Yaskawa INFORM job: DEMO_ROOF_SIDE_0625_3PAINT_25.JBI

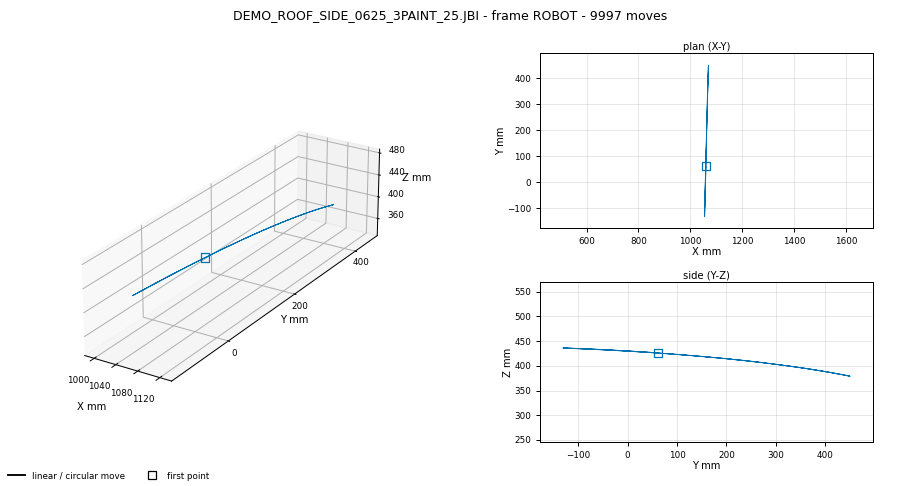
[picture p0: tool path of DEMO_ROOF_SIDE_0625_3PAINT_25.JBI in frame ROBOT, 9997 of 9997 moves have a stored position in this frame; points joined in program order, loops and branches not executed]
/JOB
//NAME DEMO_ROOF_SIDE_0625_3PAINT25
//POS
///NPOS 9997,0,0,0,0,0
///TOOL 0
///USER 0
///POSTYPE ROBOT
///RECTAN
///RCONF 1,0,0,0,0,0,0,0,0,0,0,0,0,0,0,0,0,0,0,0,0,0,0,0
C00000=1059.838,61.557,426.310,171.754,29.522,155.486
C00001=1059.832,61.309,426.327,171.753,29.519,155.486
C00002=1059.826,61.059,426.345,171.752,29.517,155.485
C00003=1059.820,60.810,426.362,171.750,29.515,155.485
C00004=1059.814,60.561,426.379,171.748,29.512,155.485
C00005=1059.807,60.311,426.396,171.747,29.509,155.484
C00006=1059.801,60.062,426.413,171.746,29.507,155.484
C00007=1059.795,59.813,426.431,171.744,29.505,155.484
C00008=1059.789,59.563,426.447,171.743,29.502,155.483
C00009=1059.783,59.314,426.465,171.741,29.500,155.483
C00010=1059.777,59.065,426.482,171.739,29.497,155.482
C00011=1059.771,58.816,426.499,171.739,29.494,155.482
C00012=1059.765,58.566,426.517,171.737,29.492,155.482
C00013=1059.758,58.317,426.534,171.735,29.489,155.481
C00014=1059.752,58.067,426.550,171.733,29.487,155.481
C00015=1059.746,57.818,426.568,171.733,29.485,155.481
C00016=1059.740,57.569,426.585,171.731,29.482,155.480
C00017=1059.734,57.319,426.602,171.729,29.479,155.480
C00018=1059.728,57.070,426.619,171.728,29.477,155.480
C00019=1059.722,56.821,426.635,171.726,29.474,155.479
C00020=1059.716,56.571,426.653,171.725,29.472,155.479
C00021=1059.710,56.322,426.670,171.723,29.470,155.478
C00022=1059.703,56.072,426.687,171.722,29.467,155.478
C00023=1059.698,55.823,426.704,171.720,29.464,155.478
C00024=1059.692,55.574,426.721,171.719,29.462,155.477
C00025=1059.685,55.324,426.738,171.718,29.459,155.477
C00026=1059.680,55.075,426.755,171.716,29.457,155.477
C00027=1059.673,54.826,426.772,171.714,29.454,155.476
C00028=1059.666,54.577,426.789,171.712,29.452,155.476
C00029=1059.661,54.327,426.806,171.712,29.449,155.475
C00030=1059.655,54.078,426.823,171.710,29.446,155.475
C00031=1059.648,53.828,426.839,171.708,29.444,155.475
C00032=1059.643,53.579,426.857,171.707,29.441,155.474
C00033=1059.637,53.330,426.873,171.706,29.439,155.474
C00034=1059.631,53.081,426.890,171.704,29.437,155.474
C00035=1059.625,52.831,426.907,171.703,29.434,155.473
C00036=1059.619,52.582,426.924,171.701,29.431,155.473
C00037=1059.613,52.333,426.941,171.700,29.429,155.473
C00038=1059.607,52.083,426.959,171.698,29.426,155.472
C00039=1059.601,51.834,426.975,171.697,29.424,155.472
C00040=1059.595,51.584,426.991,171.695,29.422,155.472
C00041=1059.589,51.335,427.009,171.693,29.419,155.471
C00042=1059.583,51.085,427.025,171.693,29.416,155.471
C00043=1059.576,50.836,427.042,171.691,29.413,155.470
C00044=1059.571,50.587,427.059,171.689,29.411,155.470
C00045=1059.565,50.338,427.076,171.688,29.409,155.470
C00046=1059.558,50.088,427.093,171.687,29.406,155.469
C00047=1059.553,49.838,427.110,171.685,29.404,155.469
C00048=1059.547,49.590,427.127,171.683,29.401,155.469
C00049=1059.541,49.340,427.143,171.682,29.398,155.468
C00050=1059.534,49.091,427.160,171.680,29.396,155.468
C00051=1059.529,48.841,427.177,171.679,29.394,155.467
C00052=1059.523,48.592,427.193,171.678,29.391,155.467
C00053=1059.517,48.343,427.210,171.676,29.388,155.467
C00054=1059.511,48.093,427.227,171.674,29.386,155.466
C00055=1059.505,47.843,427.244,171.674,29.383,155.466
C00056=1059.499,47.595,427.261,171.672,29.381,155.466
C00057=1059.493,47.345,427.277,171.670,29.378,155.465
C00058=1059.487,47.096,427.294,171.668,29.376,155.465
C00059=1059.481,46.847,427.311,171.668,29.373,155.464
C00060=1059.475,46.597,427.327,171.666,29.370,155.464
C00061=1059.468,46.313,427.346,171.664,29.368,155.464
C00062=1059.462,46.027,427.366,171.663,29.365,155.463
C00063=1059.455,45.742,427.385,171.661,29.361,155.463
C00064=1059.448,45.458,427.404,171.659,29.359,155.462
C00065=1059.442,45.208,427.420,171.658,29.356,155.462
C00066=1059.436,44.959,427.437,171.656,29.354,155.462
C00067=1059.430,44.709,427.453,171.654,29.351,155.461
C00068=1059.424,44.461,427.470,171.654,29.348,155.461
C00069=1059.419,44.211,427.487,171.652,29.346,155.461
C00070=1059.412,43.961,427.503,171.650,29.343,155.460
C00071=1059.406,43.711,427.520,171.649,29.341,155.460
C00072=1059.401,43.462,427.536,171.648,29.338,155.459
C00073=1059.394,43.213,427.553,171.646,29.336,155.459
C00074=1059.388,42.964,427.569,171.645,29.333,155.459
C00075=1059.382,42.715,427.585,171.643,29.331,155.458
C00076=1059.376,42.465,427.602,171.641,29.328,155.458
C00077=1059.370,42.215,427.618,171.640,29.326,155.458
C00078=1059.364,41.966,427.635,171.639,29.324,155.457
C00079=1059.358,41.717,427.651,171.637,29.321,155.457
C00080=1059.352,41.468,427.668,171.635,29.319,155.457
C00081=1059.346,41.218,427.684,171.635,29.316,155.456
C00082=1059.340,40.969,427.700,171.633,29.313,155.456
C00083=1059.333,40.719,427.717,171.631,29.311,155.455
C00084=1059.327,40.470,427.733,171.630,29.308,155.455
C00085=1059.322,40.220,427.750,171.628,29.306,155.455
C00086=1059.316,39.971,427.766,171.627,29.304,155.454
C00087=1059.310,39.721,427.783,171.625,29.301,155.454
C00088=1059.304,39.472,427.799,171.624,29.299,155.454
C00089=1059.298,39.223,427.815,171.622,29.296,155.453
C00090=1059.292,38.973,427.831,171.620,29.293,155.453
C00091=1059.286,38.724,427.848,171.620,29.291,155.453
C00092=1059.280,38.474,427.864,171.618,29.288,155.452
C00093=1059.274,38.225,427.880,171.616,29.286,155.452
C00094=1059.268,37.975,427.897,171.615,29.283,155.452
C00095=1059.262,37.726,427.913,171.614,29.281,155.451
C00096=1059.255,37.477,427.929,171.612,29.279,155.451
C00097=1059.249,37.228,427.945,171.610,29.276,155.450
C00098=1059.243,36.978,427.961,171.609,29.274,155.450
C00099=1059.237,36.729,427.977,171.607,29.271,155.450
C00100=1059.231,36.479,427.994,171.606,29.269,155.449
C00101=1059.224,36.230,428.010,171.605,29.266,155.449
C00102=1059.218,35.980,428.026,171.603,29.264,155.449
C00103=1059.212,35.731,428.042,171.601,29.261,155.448
C00104=1059.206,35.482,428.058,171.600,29.259,155.448
C00105=1059.200,35.232,428.075,171.599,29.256,155.448
C00106=1059.194,34.983,428.090,171.597,29.254,155.447
C00107=1059.188,34.734,428.107,171.595,29.252,155.447
C00108=1059.182,34.484,428.122,171.594,29.249,155.447
C00109=1059.176,34.235,428.138,171.593,29.247,155.446
C00110=1059.170,33.985,428.155,171.591,29.244,155.446
C00111=1059.164,33.736,428.170,171.590,29.242,155.446
C00112=1059.158,33.487,428.187,171.588,29.239,155.445
C00113=1059.152,33.238,428.203,171.586,29.237,155.445
C00114=1059.146,32.988,428.219,171.586,29.234,155.445
C00115=1059.139,32.738,428.235,171.584,29.232,155.444
C00116=1059.133,32.488,428.251,171.582,29.229,155.444
C00117=1059.127,32.239,428.267,171.580,29.227,155.444
C00118=1059.121,31.990,428.283,171.579,29.224,155.443
C00119=1059.115,31.740,428.299,171.578,29.222,155.443
C00120=1059.108,31.491,428.314,171.576,29.220,155.443
C00121=1059.103,31.241,428.331,171.575,29.217,155.442
C00122=1059.097,30.992,428.347,171.573,29.215,155.442
C00123=1059.091,30.743,428.363,171.571,29.212,155.442
C00124=1059.085,30.493,428.379,171.571,29.210,155.441
C00125=1059.078,30.209,428.397,171.569,29.207,155.441
C00126=1059.071,29.923,428.415,171.567,29.204,155.440
C00127=1059.064,29.639,428.434,171.565,29.201,155.440
C00128=1059.057,29.354,428.451,171.563,29.199,155.440
C00129=1059.051,29.105,428.468,171.562,29.196,155.439
C00130=1059.045,28.855,428.483,171.561,29.194,155.439
C00131=1059.039,28.606,428.499,171.559,29.191,155.439
C00132=1059.033,28.356,428.515,171.557,29.189,155.438
C00133=1059.027,28.106,428.531,171.556,29.186,155.438
C00134=1059.020,27.857,428.546,171.555,29.184,155.438
C00135=1059.014,27.608,428.562,171.553,29.181,155.437
C00136=1059.009,27.358,428.578,171.551,29.179,155.437
C00137=1059.002,27.109,428.594,171.550,29.177,155.437
C00138=1058.996,26.860,428.610,171.548,29.174,155.436
C00139=1058.990,26.610,428.625,171.547,29.172,155.436
C00140=1058.984,26.361,428.641,171.546,29.169,155.436
C00141=1058.977,26.111,428.657,171.544,29.167,155.435
C00142=1058.971,25.862,428.672,171.542,29.164,155.435
C00143=1058.965,25.612,428.689,171.541,29.162,155.435
C00144=1058.959,25.363,428.704,171.540,29.160,155.434
C00145=1058.953,25.113,428.720,171.538,29.158,155.434
C00146=1058.946,24.864,428.735,171.536,29.155,155.434
C00147=1058.941,24.614,428.751,171.535,29.153,155.433
C00148=1058.935,24.366,428.766,171.533,29.150,155.433
C00149=1058.929,24.116,428.782,171.532,29.148,155.432
C00150=1058.922,23.867,428.797,171.531,29.146,155.432
C00151=1058.917,23.617,428.813,171.529,29.143,155.432
C00152=1058.910,23.368,428.829,171.527,29.141,155.432
C00153=1058.904,23.118,428.844,171.526,29.138,155.431
C00154=1058.898,22.869,428.860,171.525,29.136,155.431
C00155=1058.892,22.619,428.875,171.523,29.134,155.431
C00156=1058.886,22.369,428.892,171.522,29.131,155.430
C00157=1058.880,22.120,428.907,171.520,29.129,155.430
C00158=1058.874,21.870,428.923,171.518,29.126,155.430
C00159=1058.868,21.622,428.937,171.517,29.124,155.429
C00160=1058.862,21.372,428.954,171.516,29.122,155.429
C00161=1058.856,21.123,428.969,171.514,29.119,155.429
C00162=1058.850,20.873,428.985,171.512,29.117,155.428
C00163=1058.843,20.624,429.000,171.511,29.114,155.428
C00164=1058.837,20.374,429.016,171.509,29.112,155.428
C00165=1058.831,20.125,429.031,171.508,29.109,155.427
C00166=1058.825,19.875,429.046,171.507,29.107,155.427
C00167=1058.819,19.626,429.062,171.505,29.105,155.427
C00168=1058.813,19.377,429.077,171.503,29.102,155.426
C00169=1058.807,19.127,429.093,171.502,29.100,155.426
C00170=1058.801,18.878,429.108,171.501,29.098,155.426
C00171=1058.794,18.628,429.123,171.499,29.095,155.425
C00172=1058.788,18.379,429.139,171.497,29.093,155.425
C00173=1058.782,18.129,429.154,171.496,29.090,155.425
C00174=1058.776,17.879,429.170,171.494,29.088,155.424
C00175=1058.770,17.631,429.185,171.493,29.086,155.424
C00176=1058.764,17.381,429.200,171.492,29.083,155.424
C00177=1058.758,17.131,429.216,171.490,29.081,155.423
C00178=1058.751,16.882,429.231,171.488,29.079,155.423
C00179=1058.745,16.632,429.246,171.487,29.076,155.423
C00180=1058.739,16.382,429.262,171.485,29.074,155.422
C00181=1058.733,16.134,429.277,171.484,29.071,155.422
C00182=1058.728,15.884,429.293,171.482,29.069,155.422
C00183=1058.721,15.634,429.307,171.481,29.067,155.421
C00184=1058.715,15.385,429.322,171.479,29.064,155.421
C00185=1058.709,15.135,429.339,171.477,29.062,155.421
C00186=1058.703,14.886,429.353,171.477,29.060,155.420
C00187=1058.697,14.637,429.368,171.475,29.057,155.420
C00188=1058.691,14.387,429.384,171.473,29.055,155.420
C00189=1058.684,14.104,429.401,171.472,29.052,155.419
C00190=1058.676,13.820,429.419,171.470,29.050,155.419
C00191=1058.669,13.537,429.435,171.468,29.047,155.419
C00192=1058.662,13.253,429.453,171.467,29.044,155.418
C00193=1058.656,13.004,429.468,171.465,29.042,155.418
C00194=1058.650,12.754,429.483,171.463,29.040,155.418
C00195=1058.644,12.504,429.498,171.462,29.037,155.417
C00196=1058.637,12.255,429.513,171.460,29.035,155.417
C00197=1058.631,12.005,429.528,171.458,29.033,155.417
C00198=1058.625,11.756,429.543,171.457,29.031,155.417
C00199=1058.619,11.507,429.558,171.456,29.028,155.416
C00200=1058.613,11.257,429.573,171.454,29.026,155.416
C00201=1058.606,11.007,429.588,171.452,29.023,155.416
C00202=1058.600,10.758,429.603,171.451,29.021,155.415
C00203=1058.594,10.509,429.618,171.449,29.019,155.415
C00204=1058.588,10.259,429.633,171.447,29.016,155.415
C00205=1058.581,10.010,429.648,171.447,29.014,155.414
C00206=1058.576,9.760,429.663,171.445,29.012,155.414
C00207=1058.570,9.511,429.678,171.443,29.010,155.414
C00208=1058.563,9.262,429.693,171.442,29.007,155.413
C00209=1058.557,9.012,429.708,171.440,29.005,155.413
C00210=1058.551,8.762,429.723,171.438,29.003,155.413
C00211=1058.545,8.513,429.738,171.437,29.001,155.413
C00212=1058.538,8.264,429.753,171.436,28.999,155.412
C00213=1058.532,8.014,429.768,171.434,28.996,155.412
C00214=1058.526,7.764,429.783,171.432,28.994,155.412
C00215=1058.520,7.515,429.797,171.431,28.991,155.411
C00216=1058.514,7.265,429.813,171.429,28.989,155.411
C00217=1058.508,7.016,429.828,171.428,28.987,155.411
C00218=1058.502,6.767,429.842,171.427,28.984,155.410
C00219=1058.496,6.517,429.857,171.425,28.982,155.410
C00220=1058.489,6.267,429.872,171.423,28.980,155.410
C00221=1058.483,6.018,429.887,171.421,28.978,155.410
C00222=1058.477,5.769,429.902,171.420,28.975,155.409
C00223=1058.471,5.519,429.917,171.418,28.973,155.409
C00224=1058.464,5.270,429.932,171.417,28.971,155.409
C00225=1058.459,5.020,429.946,171.416,28.969,155.408
C00226=1058.452,4.770,429.961,171.414,28.966,155.408
C00227=1058.446,4.521,429.976,171.412,28.964,155.408
C00228=1058.440,4.272,429.990,171.411,28.961,155.407
C00229=1058.434,4.022,430.005,171.409,28.959,155.407
C00230=1058.428,3.772,430.021,171.408,28.957,155.407
C00231=1058.422,3.523,430.035,171.407,28.954,155.406
C00232=1058.416,3.273,430.050,171.405,28.952,155.406
C00233=1058.410,3.025,430.065,171.403,28.950,155.406
C00234=1058.404,2.775,430.080,171.401,28.948,155.406
C00235=1058.398,2.525,430.094,171.400,28.945,155.405
C00236=1058.392,2.276,430.108,171.398,28.943,155.405
C00237=1058.386,2.026,430.123,171.397,28.941,155.405
C00238=1058.379,1.776,430.138,171.396,28.939,155.404
C00239=1058.374,1.527,430.153,171.394,28.936,155.404
C00240=1058.367,1.278,430.168,171.392,28.934,155.404
C00241=1058.362,1.028,430.182,171.391,28.931,155.403
C00242=1058.355,0.778,430.197,171.389,28.929,155.403
C00243=1058.349,0.529,430.212,171.387,28.927,155.403
C00244=1058.343,0.280,430.226,171.386,28.925,155.403
C00245=1058.337,0.030,430.241,171.385,28.922,155.402
C00246=1058.331,-0.219,430.255,171.383,28.920,155.402
C00247=1058.325,-0.469,430.270,171.381,28.918,155.402
C00248=1058.319,-0.718,430.285,171.380,28.915,155.401
C00249=1058.313,-0.968,430.299,171.378,28.913,155.401
C00250=1058.307,-1.217,430.313,171.376,28.910,155.401
C00251=1058.301,-1.467,430.328,171.376,28.908,155.400
C00252=1058.294,-1.717,430.343,171.374,28.906,155.400
C00253=1058.288,-1.998,430.360,171.372,28.903,155.400
C00254=1058.281,-2.280,430.376,171.371,28.901,155.400
C00255=1058.275,-2.561,430.392,171.368,28.898,155.399
C00256=1058.268,-2.843,430.409,171.366,28.896,155.399
C00257=1058.262,-3.092,430.423,171.365,28.893,155.398
C00258=1058.256,-3.342,430.438,171.364,28.891,155.398
C00259=1058.250,-3.592,430.452,171.362,28.889,155.398
C00260=1058.243,-3.841,430.466,171.361,28.887,155.398
C00261=1058.237,-4.091,430.481,171.359,28.885,155.397
C00262=1058.231,-4.340,430.495,171.357,28.882,155.397
C00263=1058.225,-4.590,430.510,171.356,28.880,155.397
C00264=1058.219,-4.839,430.523,171.354,28.878,155.397
C00265=1058.212,-5.089,430.538,171.352,28.876,155.396
C00266=1058.206,-5.339,430.553,171.351,28.874,155.396
C00267=1058.200,-5.588,430.567,171.350,28.872,155.396
C00268=1058.193,-5.837,430.582,171.348,28.869,155.395
C00269=1058.188,-6.087,430.595,171.346,28.867,155.395
C00270=1058.181,-6.336,430.610,171.345,28.865,155.395
C00271=1058.175,-6.586,430.624,171.343,28.863,155.395
C00272=1058.169,-6.835,430.639,171.341,28.860,155.394
C00273=1058.163,-7.085,430.652,171.339,28.858,155.394
C00274=1058.156,-7.334,430.667,171.338,28.856,155.394
C00275=1058.151,-7.584,430.681,171.337,28.854,155.394
C00276=1058.144,-7.834,430.696,171.335,28.852,155.393
C00277=1058.138,-8.083,430.709,171.334,28.850,155.393
C00278=1058.132,-8.332,430.724,171.332,28.847,155.393
C00279=1058.126,-8.582,430.738,171.330,28.845,155.392
C00280=1058.119,-8.831,430.752,171.329,28.843,155.392
C00281=1058.114,-9.081,430.766,171.327,28.841,155.392
C00282=1058.107,-9.331,430.781,171.325,28.839,155.392
C00283=1058.102,-9.580,430.795,171.323,28.836,155.391
C00284=1058.095,-9.830,430.809,171.323,28.834,155.391
C00285=1058.089,-10.079,430.823,171.321,28.832,155.391
C00286=1058.083,-10.329,430.838,171.319,28.830,155.390
C00287=1058.077,-10.578,430.851,171.318,28.828,155.390
C00288=1058.070,-10.828,430.866,171.316,28.825,155.390
C00289=1058.065,-11.077,430.880,171.314,28.823,155.390
C00290=1058.058,-11.327,430.894,171.313,28.821,155.389
C00291=1058.052,-11.576,430.908,171.311,28.819,155.389
C00292=1058.047,-11.826,430.922,171.309,28.817,155.389
C00293=1058.040,-12.075,430.936,171.308,28.815,155.389
C00294=1058.034,-12.325,430.950,171.307,28.812,155.388
C00295=1058.027,-12.575,430.964,171.305,28.810,155.388
C00296=1058.021,-12.824,430.978,171.303,28.808,155.388
C00297=1058.016,-13.073,430.992,171.302,28.806,155.387
C00298=1058.009,-13.323,431.006,171.300,28.804,155.387
C00299=1058.003,-13.572,431.021,171.298,28.801,155.387
C00300=1057.997,-13.822,431.035,171.297,28.799,155.387
C00301=1057.991,-14.072,431.048,171.295,28.797,155.387
C00302=1057.985,-14.321,431.063,171.293,28.795,155.386
C00303=1057.979,-14.571,431.077,171.292,28.793,155.386
C00304=1057.973,-14.820,431.090,171.291,28.791,155.386
C00305=1057.967,-15.070,431.105,171.289,28.789,155.385
C00306=1057.960,-15.319,431.118,171.287,28.787,155.385
C00307=1057.955,-15.569,431.132,171.286,28.784,155.385
C00308=1057.948,-15.819,431.146,171.284,28.782,155.385
C00309=1057.942,-16.068,431.160,171.282,28.780,155.384
C00310=1057.936,-16.318,431.174,171.281,28.778,155.384
C00311=1057.929,-16.567,431.187,171.279,28.776,155.384
C00312=1057.923,-16.817,431.202,171.277,28.774,155.384
C00313=1057.917,-17.066,431.215,171.275,28.772,155.383
C00314=1057.911,-17.315,431.229,171.275,28.770,155.383
C00315=1057.904,-17.565,431.243,171.273,28.767,155.383
C00316=1057.899,-17.815,431.257,171.271,28.766,155.383
C00317=1057.893,-18.069,431.271,171.270,28.764,155.382
C00318=1057.886,-18.325,431.285,171.268,28.761,155.382
C00319=1057.879,-18.579,431.299,171.266,28.759,155.382
C00320=1057.873,-18.833,431.313,171.265,28.757,155.382
C00321=1057.867,-19.083,431.326,171.263,28.755,155.381
C00322=1057.861,-19.333,431.341,171.261,28.753,155.381
C00323=1057.855,-19.582,431.354,171.259,28.751,155.381
C00324=1057.849,-19.832,431.368,171.258,28.749,155.381
C00325=1057.842,-20.082,431.381,171.256,28.746,155.380
C00326=1057.836,-20.331,431.395,171.254,28.744,155.380
C00327=1057.830,-20.580,431.409,171.253,28.743,155.380
C00328=1057.824,-20.830,431.423,171.251,28.740,155.380
C00329=1057.818,-21.079,431.437,171.250,28.738,155.379
C00330=1057.812,-21.329,431.450,171.248,28.736,155.379
C00331=1057.805,-21.579,431.464,171.247,28.734,155.379
C00332=1057.800,-21.828,431.478,171.245,28.732,155.379
C00333=1057.793,-22.078,431.491,171.243,28.730,155.378
C00334=1057.787,-22.328,431.504,171.242,28.728,155.378
C00335=1057.781,-22.577,431.518,171.240,28.726,155.378
C00336=1057.775,-22.826,431.532,171.238,28.724,155.378
C00337=1057.769,-23.076,431.545,171.236,28.722,155.377
C00338=1057.763,-23.326,431.559,171.235,28.719,155.377
C00339=1057.756,-23.575,431.572,171.233,28.717,155.377
C00340=1057.751,-23.825,431.586,171.231,28.715,155.377
C00341=1057.745,-24.074,431.599,171.230,28.713,155.376
C00342=1057.738,-24.324,431.613,171.228,28.711,155.376
C00343=1057.732,-24.574,431.627,171.226,28.709,155.376
C00344=1057.726,-24.823,431.640,171.226,28.707,155.376
C00345=1057.720,-25.072,431.654,171.224,28.705,155.375
C00346=1057.714,-25.322,431.668,171.222,28.703,155.375
C00347=1057.708,-25.572,431.681,171.220,28.701,155.375
C00348=1057.701,-25.821,431.694,171.219,28.699,155.375
C00349=1057.696,-26.070,431.708,171.217,28.697,155.375
C00350=1057.689,-26.320,431.722,171.215,28.695,155.374
C00351=1057.683,-26.570,431.735,171.214,28.693,155.374
C00352=1057.677,-26.819,431.749,171.212,28.690,155.374
C00353=1057.671,-27.069,431.762,171.210,28.689,155.374
C00354=1057.665,-27.318,431.775,171.208,28.686,155.373
C00355=1057.659,-27.568,431.788,171.207,28.685,155.373
C00356=1057.652,-27.818,431.802,171.205,28.683,155.373
C00357=1057.646,-28.067,431.815,171.203,28.680,155.373
C00358=1057.640,-28.316,431.828,171.202,28.679,155.372
C00359=1057.634,-28.566,431.842,171.200,28.677,155.372
C00360=1057.628,-28.816,431.855,171.198,28.675,155.372
C00361=1057.621,-29.090,431.870,171.196,28.673,155.372
C00362=1057.614,-29.365,431.885,171.195,28.670,155.372
C00363=1057.607,-29.640,431.899,171.193,28.668,155.371
C00364=1057.599,-29.916,431.914,171.191,28.666,155.371
C00365=1057.594,-30.166,431.927,171.190,28.664,155.371
C00366=1057.588,-30.415,431.940,171.188,28.662,155.371
C00367=1057.582,-30.664,431.953,171.186,28.660,155.370
C00368=1057.576,-30.914,431.967,171.185,28.658,155.370
C00369=1057.569,-31.164,431.980,171.183,28.656,155.370
C00370=1057.563,-31.413,431.993,171.181,28.654,155.370
C00371=1057.557,-31.663,432.006,171.179,28.652,155.369
C00372=1057.550,-31.912,432.019,171.178,28.651,155.369
C00373=1057.545,-32.162,432.032,171.176,28.648,155.369
C00374=1057.538,-32.411,432.045,171.174,28.647,155.369
C00375=1057.532,-32.661,432.059,171.173,28.644,155.369
C00376=1057.526,-32.911,432.073,171.171,28.642,155.368
C00377=1057.520,-33.161,432.085,171.169,28.641,155.368
C00378=1057.514,-33.410,432.099,171.167,28.638,155.368
C00379=1057.508,-33.659,432.112,171.166,28.637,155.368
C00380=1057.502,-33.909,432.124,171.164,28.634,155.368
C00381=1057.494,-34.188,432.140,171.162,28.632,155.367
C00382=1057.487,-34.467,432.154,171.161,28.631,155.367
C00383=1057.481,-34.747,432.168,171.159,28.628,155.367
C00384=1057.474,-35.026,432.183,171.157,28.626,155.367
C00385=1057.468,-35.275,432.196,171.156,28.624,155.366
C00386=1057.461,-35.525,432.209,171.154,28.622,155.366
C00387=1057.455,-35.775,432.223,171.152,28.620,155.366
C00388=1057.449,-36.025,432.235,171.150,28.618,155.366
C00389=1057.443,-36.274,432.248,171.149,28.616,155.365
C00390=1057.437,-36.524,432.261,171.147,28.615,155.365
C00391=1057.431,-36.773,432.274,171.145,28.612,155.365
C00392=1057.425,-37.022,432.288,171.143,28.611,155.365
C00393=1057.419,-37.272,432.300,171.142,28.608,155.365
C00394=1057.413,-37.522,432.314,171.140,28.607,155.364
C00395=1057.407,-37.772,432.327,171.138,28.605,155.364
C00396=1057.401,-38.021,432.340,171.137,28.603,155.364
C00397=1057.395,-38.271,432.352,171.135,28.601,155.364
C00398=1057.389,-38.520,432.366,171.133,28.599,155.364
C00399=1057.383,-38.770,432.378,171.131,28.597,155.363
C00400=1057.376,-39.020,432.391,171.130,28.595,155.363
C00401=1057.370,-39.269,432.404,171.128,28.594,155.363
C00402=1057.363,-39.519,432.417,171.126,28.591,155.363
C00403=1057.357,-39.769,432.430,171.125,28.590,155.363
C00404=1057.351,-40.018,432.443,171.123,28.588,155.362
C00405=1057.345,-40.267,432.455,171.121,28.586,155.362
C00406=1057.338,-40.517,432.468,171.119,28.584,155.362
C00407=1057.333,-40.767,432.481,171.118,28.583,155.362
C00408=1057.327,-41.016,432.493,171.116,28.580,155.362
C00409=1057.320,-41.266,432.506,171.114,28.579,155.362
C00410=1057.314,-41.516,432.519,171.112,28.577,155.361
C00411=1057.308,-41.765,432.532,171.111,28.575,155.361
C00412=1057.302,-42.014,432.544,171.109,28.573,155.361
C00413=1057.296,-42.264,432.557,171.107,28.571,155.361
C00414=1057.289,-42.514,432.570,171.106,28.569,155.361
C00415=1057.284,-42.763,432.583,171.104,28.568,155.360
C00416=1057.277,-43.012,432.595,171.102,28.566,155.360
C00417=1057.271,-43.262,432.608,171.100,28.564,155.360
C00418=1057.265,-43.512,432.620,171.099,28.562,155.360
C00419=1057.259,-43.761,432.634,171.097,28.560,155.360
C00420=1057.252,-44.011,432.646,171.095,28.558,155.359
C00421=1057.246,-44.261,432.658,171.093,28.557,155.359
C00422=1057.240,-44.510,432.671,171.092,28.555,155.359
C00423=1057.234,-44.760,432.684,171.090,28.553,155.359
C00424=1057.228,-45.010,432.697,171.088,28.551,155.359
C00425=1057.221,-45.259,432.709,171.087,28.549,155.359
C00426=1057.215,-45.509,432.722,171.085,28.548,155.358
C00427=1057.209,-45.759,432.734,171.083,28.546,155.358
C00428=1057.203,-46.009,432.747,171.081,28.544,155.358
C00429=1057.196,-46.257,432.760,171.080,28.542,155.358
C00430=1057.190,-46.507,432.772,171.078,28.541,155.358
C00431=1057.185,-46.757,432.785,171.076,28.538,155.357
C00432=1057.179,-47.007,432.797,171.074,28.537,155.357
C00433=1057.172,-47.256,432.810,171.073,28.535,155.357
C00434=1057.166,-47.506,432.823,171.071,28.533,155.357
C00435=1057.160,-47.756,432.835,171.069,28.531,155.357
C00436=1057.154,-48.006,432.848,171.067,28.530,155.357
C00437=1057.147,-48.255,432.860,171.066,28.528,155.356
C00438=1057.142,-48.504,432.872,171.064,28.526,155.356
C00439=1057.136,-48.754,432.885,171.062,28.524,155.356
C00440=1057.130,-49.004,432.898,171.061,28.522,155.356
C00441=1057.123,-49.253,432.910,171.059,28.521,155.356
C00442=1057.117,-49.503,432.922,171.057,28.519,155.356
C00443=1057.111,-49.752,432.935,171.055,28.517,155.355
C00444=1057.104,-50.002,432.947,171.054,28.515,155.355
C00445=1057.098,-50.282,432.961,171.052,28.514,155.355
C00446=1057.091,-50.561,432.975,171.050,28.511,155.355
C00447=1057.084,-50.842,432.989,171.047,28.509,155.355
C00448=1057.077,-51.121,433.003,171.046,28.508,155.354
C00449=1057.071,-51.370,433.015,171.044,28.506,155.354
C00450=1057.065,-51.620,433.027,171.042,28.505,155.354
C00451=1057.058,-51.870,433.039,171.040,28.503,155.354
C00452=1057.052,-52.120,433.052,171.039,28.501,155.354
C00453=1057.045,-52.369,433.064,171.037,28.500,155.354
C00454=1057.039,-52.619,433.076,171.035,28.498,155.354
C00455=1057.033,-52.869,433.088,171.033,28.496,155.353
C00456=1057.026,-53.118,433.100,171.032,28.495,155.353
C00457=1057.021,-53.367,433.112,171.030,28.493,155.353
C00458=1057.014,-53.617,433.124,171.028,28.491,155.353
C00459=1057.008,-53.867,433.137,171.027,28.490,155.353
C00460=1057.002,-54.116,433.149,171.025,28.488,155.353
C00461=1056.995,-54.366,433.161,171.023,28.486,155.353
C00462=1056.989,-54.616,433.173,171.021,28.485,155.352
C00463=1056.982,-54.865,433.185,171.020,28.483,155.352
C00464=1056.977,-55.115,433.198,171.018,28.481,155.352
C00465=1056.971,-55.364,433.209,171.015,28.480,155.352
C00466=1056.964,-55.614,433.221,171.013,28.478,155.352
C00467=1056.958,-55.864,433.234,171.012,28.476,155.352
C00468=1056.951,-56.113,433.246,171.010,28.475,155.352
C00469=1056.945,-56.363,433.258,171.008,28.473,155.351
C00470=1056.939,-56.613,433.270,171.006,28.471,155.351
C00471=1056.932,-56.862,433.282,171.005,28.470,155.351
C00472=1056.927,-57.111,433.295,171.003,28.468,155.351
C00473=1056.920,-57.361,433.307,171.001,28.466,155.351
C00474=1056.914,-57.611,433.318,170.999,28.465,155.351
C00475=1056.908,-57.861,433.330,170.997,28.464,155.351
C00476=1056.901,-58.111,433.342,170.996,28.462,155.350
C00477=1056.895,-58.360,433.354,170.994,28.460,155.350
C00478=1056.889,-58.609,433.366,170.992,28.459,155.350
C00479=1056.883,-58.859,433.378,170.990,28.457,155.350
C00480=1056.877,-59.109,433.391,170.989,28.455,155.350
C00481=1056.870,-59.358,433.403,170.987,28.454,155.350
C00482=1056.864,-59.608,433.414,170.985,28.452,155.350
C00483=1056.858,-59.858,433.426,170.984,28.451,155.349
C00484=1056.852,-60.107,433.438,170.982,28.449,155.349
C00485=1056.845,-60.357,433.450,170.980,28.448,155.349
C00486=1056.840,-60.606,433.462,170.978,28.446,155.349
C00487=1056.834,-60.856,433.474,170.976,28.445,155.349
C00488=1056.827,-61.106,433.486,170.975,28.443,155.349
C00489=1056.821,-61.356,433.498,170.972,28.441,155.349
C00490=1056.815,-61.605,433.510,170.970,28.439,155.349
C00491=1056.809,-61.855,433.521,170.969,28.438,155.348
C00492=1056.803,-62.105,433.534,170.967,28.436,155.348
C00493=1056.796,-62.354,433.546,170.965,28.435,155.348
C00494=1056.790,-62.603,433.557,170.963,28.433,155.348
C00495=1056.784,-62.854,433.569,170.961,28.432,155.348
C00496=1056.778,-63.103,433.581,170.960,28.430,155.348
C00497=1056.771,-63.353,433.593,170.958,28.428,155.348
C00498=1056.765,-63.602,433.604,170.956,28.427,155.347
C00499=1056.759,-63.852,433.616,170.954,28.426,155.347
C00500=1056.753,-64.102,433.628,170.953,28.424,155.347
C00501=1056.747,-64.351,433.640,170.951,28.422,155.347
C00502=1056.741,-64.601,433.652,170.949,28.421,155.347
C00503=1056.735,-64.851,433.664,170.947,28.419,155.347
C00504=1056.728,-65.100,433.675,170.946,28.418,155.347
C00505=1056.723,-65.350,433.687,170.944,28.416,155.347
C00506=1056.716,-65.600,433.699,170.942,28.415,155.347
C00507=1056.710,-65.849,433.710,170.940,28.413,155.346
C00508=1056.704,-66.099,433.722,170.938,28.411,155.346
C00509=1056.697,-66.380,433.735,170.936,28.410,155.346
C00510=1056.690,-66.660,433.749,170.934,28.408,155.346
C00511=1056.683,-66.942,433.762,170.932,28.406,155.346
C00512=1056.676,-67.223,433.775,170.930,28.404,155.346
C00513=1056.671,-67.472,433.787,170.928,28.403,155.346
C00514=1056.665,-67.722,433.798,170.926,28.402,155.346
C00515=1056.658,-67.972,433.810,170.924,28.400,155.345
C00516=1056.652,-68.221,433.821,170.923,28.398,155.345
C00517=1056.646,-68.471,433.834,170.921,28.397,155.345
C00518=1056.641,-68.721,433.845,170.919,28.396,155.345
C00519=1056.634,-68.970,433.856,170.917,28.394,155.345
C00520=1056.628,-69.220,433.868,170.916,28.392,155.345
C00521=1056.622,-69.470,433.880,170.914,28.391,155.345
C00522=1056.616,-69.720,433.891,170.912,28.390,155.345
C00523=1056.610,-69.969,433.903,170.910,28.388,155.344
C00524=1056.604,-70.219,433.914,170.909,28.386,155.344
C00525=1056.598,-70.468,433.926,170.906,28.385,155.344
C00526=1056.592,-70.718,433.937,170.904,28.383,155.344
C00527=1056.586,-70.967,433.949,170.902,28.382,155.344
C00528=1056.580,-71.217,433.960,170.900,28.381,155.344
C00529=1056.574,-71.467,433.973,170.899,28.379,155.344
C00530=1056.568,-71.717,433.984,170.897,28.377,155.344
C00531=1056.561,-71.966,433.996,170.895,28.376,155.344
C00532=1056.555,-72.216,434.007,170.893,28.375,155.344
C00533=1056.549,-72.465,434.018,170.892,28.373,155.343
C00534=1056.544,-72.715,434.030,170.890,28.371,155.343
C00535=1056.537,-72.965,434.041,170.888,28.370,155.343
C00536=1056.531,-73.214,434.053,170.886,28.369,155.343
C00537=1056.525,-73.464,434.064,170.885,28.367,155.343
C00538=1056.519,-73.714,434.075,170.883,28.366,155.343
C00539=1056.513,-73.964,434.087,170.881,28.364,155.343
C00540=1056.508,-74.213,434.098,170.878,28.363,155.343
C00541=1056.501,-74.463,434.110,170.876,28.361,155.343
C00542=1056.495,-74.712,434.121,170.875,28.360,155.343
C00543=1056.489,-74.962,434.132,170.873,28.359,155.342
C00544=1056.482,-75.212,434.144,170.871,28.358,155.342
C00545=1056.477,-75.462,434.155,170.869,28.356,155.342
C00546=1056.470,-75.712,434.167,170.868,28.355,155.342
C00547=1056.465,-75.961,434.177,170.866,28.353,155.342
C00548=1056.458,-76.211,434.189,170.864,28.352,155.342
C00549=1056.451,-76.460,434.200,170.862,28.350,155.342
C00550=1056.445,-76.710,434.211,170.860,28.349,155.342
C00551=1056.439,-76.959,434.222,170.859,28.348,155.342
C00552=1056.433,-77.209,434.234,170.857,28.347,155.342
C00553=1056.427,-77.459,434.245,170.854,28.345,155.342
C00554=1056.421,-77.709,434.256,170.852,28.344,155.342
C00555=1056.415,-77.958,434.267,170.851,28.342,155.341
C00556=1056.408,-78.208,434.279,170.849,28.341,155.341
C00557=1056.402,-78.457,434.290,170.847,28.340,155.341
C00558=1056.396,-78.708,434.301,170.845,28.338,155.341
C00559=1056.390,-78.957,434.312,170.843,28.337,155.341
C00560=1056.384,-79.206,434.323,170.842,28.336,155.341
C00561=1056.378,-79.456,434.335,170.840,28.335,155.341
C00562=1056.372,-79.706,434.345,170.838,28.334,155.341
C00563=1056.366,-79.956,434.357,170.836,28.332,155.341
C00564=1056.359,-80.205,434.367,170.833,28.331,155.341
C00565=1056.353,-80.455,434.378,170.832,28.330,155.341
C00566=1056.347,-80.704,434.390,170.830,28.328,155.341
C00567=1056.341,-80.954,434.401,170.828,28.327,155.341
C00568=1056.334,-81.203,434.411,170.826,28.326,155.341
C00569=1056.328,-81.454,434.423,170.824,28.325,155.341
C00570=1056.322,-81.703,434.433,170.823,28.323,155.340
C00571=1056.316,-81.953,434.445,170.821,28.322,155.340
C00572=1056.309,-82.203,434.455,170.819,28.321,155.340
C00573=1056.302,-82.487,434.468,170.816,28.320,155.340
C00574=1056.295,-82.769,434.480,170.815,28.318,155.340
C00575=1056.288,-83.052,434.492,170.813,28.317,155.340
C00576=1056.281,-83.336,434.505,170.810,28.315,155.340
C00577=1056.275,-83.585,434.516,170.808,28.314,155.340
C00578=1056.268,-83.835,434.527,170.806,28.313,155.340
C00579=1056.263,-84.084,434.538,170.805,28.312,155.340
C00580=1056.256,-84.334,434.548,170.803,28.311,155.340
C00581=1056.250,-84.584,434.560,170.801,28.309,155.340
C00582=1056.244,-84.833,434.570,170.799,28.308,155.340
C00583=1056.237,-85.083,434.581,170.796,28.307,155.340
C00584=1056.231,-85.333,434.592,170.795,28.306,155.340
C00585=1056.225,-85.582,434.603,170.793,28.305,155.340
C00586=1056.219,-85.832,434.614,170.791,28.304,155.340
C00587=1056.213,-86.082,434.624,170.789,28.302,155.340
C00588=1056.207,-86.332,434.635,170.787,28.301,155.340
C00589=1056.201,-86.582,434.646,170.786,28.300,155.339
C00590=1056.194,-86.831,434.656,170.784,28.299,155.339
C00591=1056.188,-87.081,434.667,170.782,28.298,155.339
C00592=1056.182,-87.331,434.678,170.780,28.297,155.339
C00593=1056.176,-87.580,434.688,170.777,28.295,155.339
C00594=1056.169,-87.830,434.700,170.776,28.294,155.339
C00595=1056.164,-88.080,434.711,170.774,28.293,155.339
C00596=1056.157,-88.329,434.721,170.772,28.292,155.339
C00597=1056.151,-88.579,434.732,170.770,28.291,155.339
C00598=1056.145,-88.828,434.743,170.768,28.289,155.339
C00599=1056.139,-89.078,434.753,170.766,28.288,155.339
C00600=1056.133,-89.328,434.764,170.765,28.287,155.339
C00601=1056.127,-89.578,434.775,170.763,28.286,155.339
C00602=1056.120,-89.827,434.785,170.760,28.285,155.339
C00603=1056.114,-90.077,434.796,170.758,28.284,155.339
C00604=1056.108,-90.326,434.806,170.756,28.283,155.339
C00605=1056.102,-90.576,434.817,170.755,28.281,155.339
C00606=1056.096,-90.827,434.828,170.753,28.280,155.339
C00607=1056.089,-91.076,434.838,170.751,28.279,155.339
C00608=1056.084,-91.325,434.849,170.749,28.278,155.339
C00609=1056.078,-91.575,434.860,170.747,28.277,155.339
C00610=1056.071,-91.825,434.871,170.746,28.276,155.339
C00611=1056.065,-92.075,434.881,170.744,28.275,155.339
C00612=1056.060,-92.324,434.892,170.741,28.274,155.339
C00613=1056.053,-92.574,434.902,170.739,28.273,155.339
C00614=1056.047,-92.824,434.913,170.737,28.271,155.339
C00615=1056.041,-93.074,434.923,170.735,28.270,155.339
C00616=1056.035,-93.323,434.934,170.734,28.269,155.339
C00617=1056.029,-93.573,434.944,170.732,28.268,155.339
C00618=1056.022,-93.822,434.955,170.730,28.267,155.339
C00619=1056.017,-94.073,434.965,170.728,28.266,155.338
C00620=1056.010,-94.322,434.976,170.726,28.265,155.338
C00621=1056.004,-94.571,434.986,170.724,28.264,155.338
C00622=1055.999,-94.821,434.997,170.722,28.263,155.338
C00623=1055.992,-95.071,435.007,170.720,28.262,155.338
C00624=1055.986,-95.321,435.018,170.718,28.261,155.338
C00625=1055.980,-95.570,435.028,170.716,28.260,155.338
C00626=1055.974,-95.820,435.039,170.714,28.258,155.338
C00627=1055.968,-96.069,435.049,170.713,28.257,155.338
C00628=1055.962,-96.320,435.059,170.711,28.256,155.338
C00629=1055.956,-96.569,435.070,170.709,28.255,155.338
C00630=1055.949,-96.819,435.081,170.706,28.254,155.338
C00631=1055.944,-97.069,435.091,170.704,28.253,155.338
C00632=1055.938,-97.318,435.101,170.703,28.252,155.338
C00633=1055.931,-97.568,435.112,170.701,28.251,155.338
C00634=1055.925,-97.818,435.122,170.699,28.250,155.338
C00635=1055.919,-98.067,435.133,170.697,28.249,155.338
C00636=1055.913,-98.317,435.142,170.695,28.248,155.338
C00637=1055.906,-98.603,435.155,170.692,28.247,155.338
C00638=1055.899,-98.888,435.166,170.691,28.246,155.338
C00639=1055.892,-99.173,435.178,170.688,28.245,155.338
C00640=1055.885,-99.459,435.190,170.686,28.244,155.338
C00641=1055.879,-99.709,435.199,170.684,28.243,155.338
C00642=1055.872,-99.958,435.209,170.682,28.242,155.338
C00643=1055.866,-100.208,435.221,170.680,28.242,155.338
C00644=1055.860,-100.458,435.230,170.679,28.240,155.338
C00645=1055.854,-100.708,435.240,170.676,28.239,155.338
C00646=1055.848,-100.957,435.251,170.674,28.238,155.338
C00647=1055.842,-101.207,435.260,170.672,28.238,155.338
C00648=1055.835,-101.456,435.271,170.670,28.237,155.338
C00649=1055.830,-101.706,435.281,170.668,28.236,155.338
C00650=1055.823,-101.956,435.291,170.667,28.235,155.338
C00651=1055.817,-102.206,435.301,170.665,28.234,155.338
C00652=1055.811,-102.456,435.312,170.663,28.233,155.338
C00653=1055.805,-102.705,435.321,170.660,28.232,155.338
C00654=1055.798,-102.955,435.332,170.658,28.231,155.338
C00655=1055.793,-103.205,435.342,170.656,28.230,155.338
C00656=1055.787,-103.455,435.351,170.655,28.230,155.338
C00657=1055.780,-103.704,435.362,170.653,28.229,155.338
C00658=1055.773,-103.954,435.372,170.651,28.228,155.338
C00659=1055.768,-104.204,435.383,170.649,28.227,155.339
C00660=1055.762,-104.453,435.392,170.647,28.226,155.338
C00661=1055.755,-104.703,435.402,170.644,28.225,155.338
C00662=1055.750,-104.953,435.413,170.642,28.224,155.339
C00663=1055.743,-105.203,435.422,170.641,28.223,155.339
C00664=1055.737,-105.452,435.432,170.639,28.223,155.339
C00665=1055.731,-105.702,435.442,170.637,28.222,155.339
C00666=1055.725,-105.952,435.452,170.635,28.221,155.339
C00667=1055.719,-106.201,435.462,170.633,28.220,155.339
C00668=1055.713,-106.451,435.472,170.631,28.219,155.339
C00669=1055.707,-106.700,435.482,170.629,28.218,155.339
C00670=1055.701,-106.951,435.492,170.627,28.217,155.339
C00671=1055.695,-107.200,435.502,170.625,28.217,155.339
C00672=1055.688,-107.450,435.512,170.623,28.216,155.339
C00673=1055.682,-107.700,435.521,170.621,28.215,155.339
C00674=1055.676,-107.950,435.531,170.619,28.214,155.339
C00675=1055.670,-108.199,435.542,170.617,28.214,155.339
C00676=1055.664,-108.449,435.551,170.615,28.213,155.339
C00677=1055.657,-108.699,435.561,170.613,28.212,155.339
C00678=1055.651,-108.949,435.571,170.611,28.211,155.339
C00679=1055.645,-109.198,435.581,170.609,28.211,155.339
C00680=1055.639,-109.448,435.590,170.607,28.210,155.339
C00681=1055.632,-109.697,435.600,170.605,28.209,155.339
C00682=1055.626,-109.947,435.610,170.603,28.209,155.339
C00683=1055.621,-110.197,435.620,170.602,28.208,155.339
C00684=1055.614,-110.447,435.630,170.599,28.207,155.339
C00685=1055.608,-110.696,435.640,170.597,28.206,155.339
C00686=1055.602,-110.946,435.649,170.595,28.205,155.339
C00687=1055.596,-111.196,435.659,170.593,28.205,155.339
C00688=1055.590,-111.446,435.668,170.591,28.204,155.339
C00689=1055.583,-111.696,435.678,170.589,28.203,155.340
C00690=1055.577,-111.945,435.688,170.587,28.202,155.340
C00691=1055.571,-112.195,435.698,170.585,28.202,155.340
C00692=1055.565,-112.444,435.707,170.583,28.201,155.340
C00693=1055.558,-112.694,435.717,170.581,28.200,155.340
C00694=1055.553,-112.944,435.727,170.579,28.200,155.340
C00695=1055.547,-113.194,435.737,170.577,28.199,155.340
C00696=1055.541,-113.444,435.746,170.575,28.198,155.340
C00697=1055.535,-113.694,435.756,170.573,28.198,155.340
C00698=1055.528,-113.943,435.765,170.571,28.197,155.340
C00699=1055.522,-114.193,435.775,170.569,28.196,155.340
C00700=1055.516,-114.442,435.785,170.567,28.195,155.340
C00701=1055.509,-114.727,435.795,170.565,28.195,155.340
C00702=1055.502,-115.010,435.806,170.562,28.194,155.340
C00703=1055.495,-115.295,435.818,170.560,28.193,155.340
C00704=1055.488,-115.579,435.828,170.558,28.193,155.340
C00705=1055.482,-115.829,435.838,170.555,28.192,155.341
C00706=1055.476,-116.078,435.847,170.554,28.191,155.341
C00707=1055.470,-116.328,435.857,170.552,28.191,155.341
C00708=1055.464,-116.578,435.866,170.550,28.190,155.341
C00709=1055.457,-116.828,435.876,170.548,28.190,155.341
C00710=1055.452,-117.077,435.885,170.546,28.189,155.341
C00711=1055.446,-117.327,435.895,170.544,28.188,155.341
C00712=1055.440,-117.576,435.904,170.541,28.187,155.341
C00713=1055.433,-117.826,435.913,170.539,28.187,155.341
C00714=1055.426,-118.076,435.923,170.538,28.186,155.341
C00715=1055.420,-118.326,435.932,170.536,28.186,155.341
C00716=1055.414,-118.575,435.942,170.534,28.185,155.341
C00717=1055.408,-118.825,435.951,170.532,28.184,155.341
C00718=1055.402,-119.075,435.961,170.530,28.184,155.341
C00719=1055.396,-119.325,435.970,170.527,28.183,155.342
C00720=1055.390,-119.574,435.980,170.525,28.183,155.342
C00721=1055.384,-119.824,435.989,170.523,28.182,155.342
C00722=1055.378,-120.074,435.998,170.521,28.182,155.342
C00723=1055.371,-120.324,436.007,170.520,28.181,155.342
C00724=1055.365,-120.573,436.017,170.518,28.180,155.342
C00725=1055.359,-120.823,436.026,170.516,28.180,155.342
C00726=1055.353,-121.073,436.036,170.513,28.179,155.342
C00727=1055.347,-121.322,436.045,170.511,28.179,155.342
C00728=1055.341,-121.572,436.055,170.509,28.178,155.342
C00729=1055.335,-121.822,436.063,170.507,28.178,155.342
C00730=1055.329,-122.072,436.073,170.505,28.177,155.342
C00731=1055.322,-122.322,436.082,170.503,28.177,155.342
C00732=1055.316,-122.571,436.092,170.502,28.177,155.343
C00733=1055.310,-122.820,436.101,170.499,28.176,155.343
C00734=1055.304,-123.071,436.110,170.497,28.175,155.343
C00735=1055.298,-123.321,436.119,170.495,28.175,155.343
C00736=1055.292,-123.570,436.129,170.493,28.174,155.343
C00737=1055.285,-123.820,436.138,170.491,28.174,155.343
C00738=1055.279,-124.070,436.147,170.489,28.174,155.343
C00739=1055.274,-124.319,436.156,170.487,28.173,155.343
C00740=1055.267,-124.569,436.165,170.485,28.173,155.343
C00741=1055.261,-124.819,436.175,170.483,28.172,155.343
C00742=1055.255,-125.069,436.183,170.481,28.171,155.344
C00743=1055.248,-125.319,436.193,170.479,28.171,155.344
C00744=1055.243,-125.568,436.202,170.477,28.171,155.344
C00745=1055.236,-125.818,436.211,170.475,28.170,155.344
C00746=1055.230,-126.068,436.220,170.473,28.170,155.344
C00747=1055.224,-126.318,436.229,170.470,28.170,155.344
C00748=1055.218,-126.568,436.239,170.468,28.169,155.344
C00749=1055.212,-126.817,436.247,170.466,28.169,155.344
C00750=1055.206,-127.067,436.256,170.464,28.168,155.344
C00751=1055.199,-127.317,436.266,170.462,28.168,155.344
C00752=1055.193,-127.567,436.274,170.461,28.167,155.345
C00753=1055.187,-127.816,436.283,170.459,28.167,155.345
C00754=1055.182,-128.066,436.293,170.457,28.166,155.345
C00755=1055.178,-128.316,436.303,170.455,28.165,155.345
C00756=1055.175,-128.566,436.314,170.453,28.163,155.344
C00757=1055.174,-128.817,436.325,170.452,28.161,155.344
C00758=1055.174,-129.067,436.338,170.450,28.157,155.344
C00759=1055.174,-129.318,436.351,170.449,28.154,155.343
C00760=1055.176,-129.567,436.364,170.448,28.150,155.343
C00761=1055.179,-129.819,436.379,170.447,28.145,155.342
C00762=1055.184,-130.070,436.394,170.447,28.140,155.341
C00763=1055.190,-130.321,436.410,170.445,28.135,155.340
C00764=1055.196,-130.571,436.427,170.445,28.128,155.339
C00765=1054.825,-130.594,436.216,170.397,28.295,155.372
C00766=1054.818,-130.344,436.200,170.399,28.301,155.373
C00767=1054.813,-130.093,436.184,170.399,28.307,155.374
C00768=1054.808,-129.843,436.169,170.399,28.312,155.375
C00769=1054.804,-129.591,436.155,170.400,28.316,155.376
C00770=1054.802,-129.341,436.141,170.401,28.320,155.376
C00771=1054.801,-129.091,436.128,170.402,28.324,155.377
C00772=1054.802,-128.840,436.116,170.404,28.327,155.377
C00773=1054.804,-128.590,436.104,170.405,28.329,155.378
C00774=1054.806,-128.339,436.093,170.407,28.331,155.378
C00775=1054.810,-128.089,436.083,170.409,28.333,155.378
C00776=1054.815,-127.840,436.073,170.411,28.333,155.378
C00777=1054.821,-127.589,436.064,170.413,28.334,155.378
C00778=1054.828,-127.340,436.055,170.415,28.334,155.378
C00779=1054.833,-127.091,436.046,170.417,28.335,155.378
C00780=1054.839,-126.840,436.037,170.419,28.335,155.377
C00781=1054.846,-126.591,436.028,170.421,28.336,155.377
C00782=1054.852,-126.341,436.018,170.423,28.336,155.377
C00783=1054.858,-126.091,436.010,170.425,28.336,155.377
C00784=1054.863,-125.841,436.000,170.427,28.336,155.377
C00785=1054.870,-125.592,435.991,170.429,28.337,155.377
C00786=1054.876,-125.342,435.983,170.431,28.337,155.377
C00787=1054.882,-125.092,435.973,170.433,28.338,155.377
C00788=1054.889,-124.842,435.964,170.436,28.338,155.377
C00789=1054.895,-124.593,435.955,170.438,28.339,155.376
C00790=1054.901,-124.343,435.946,170.440,28.339,155.376
C00791=1054.907,-124.093,435.936,170.441,28.340,155.376
C00792=1054.913,-123.843,435.927,170.443,28.340,155.376
C00793=1054.920,-123.593,435.919,170.445,28.341,155.376
C00794=1054.925,-123.344,435.909,170.447,28.341,155.376
C00795=1054.931,-123.094,435.900,170.450,28.342,155.376
C00796=1054.938,-122.844,435.890,170.452,28.342,155.376
C00797=1054.944,-122.595,435.881,170.454,28.343,155.376
C00798=1054.950,-122.344,435.872,170.456,28.343,155.376
C00799=1054.957,-122.095,435.863,170.458,28.344,155.376
C00800=1054.962,-121.846,435.854,170.460,28.344,155.376
C00801=1054.968,-121.596,435.844,170.462,28.345,155.375
C00802=1054.974,-121.346,435.834,170.464,28.345,155.375
C00803=1054.981,-121.096,435.825,170.466,28.346,155.375
C00804=1054.987,-120.846,435.816,170.468,28.346,155.375
C00805=1054.993,-120.596,435.806,170.470,28.347,155.375
C00806=1054.998,-120.347,435.797,170.472,28.347,155.375
C00807=1055.005,-120.097,435.788,170.474,28.347,155.375
C00808=1055.011,-119.848,435.779,170.477,28.348,155.375
C00809=1055.018,-119.598,435.769,170.479,28.349,155.375
C00810=1055.024,-119.348,435.760,170.480,28.350,155.375
C00811=1055.030,-119.098,435.751,170.482,28.350,155.375
C00812=1055.036,-118.848,435.741,170.484,28.351,155.374
C00813=1055.042,-118.598,435.732,170.486,28.351,155.374
C00814=1055.047,-118.349,435.722,170.488,28.351,155.374
C00815=1055.054,-118.099,435.713,170.491,28.352,155.374
C00816=1055.060,-117.849,435.703,170.493,28.353,155.374
C00817=1055.067,-117.600,435.694,170.495,28.354,155.374
C00818=1055.073,-117.350,435.685,170.497,28.354,155.374
C00819=1055.079,-117.100,435.675,170.498,28.355,155.374
C00820=1055.085,-116.850,435.666,170.500,28.355,155.374
C00821=1055.091,-116.601,435.656,170.502,28.355,155.374
C00822=1055.098,-116.351,435.646,170.505,28.357,155.374
C00823=1055.104,-116.101,435.637,170.507,28.357,155.374
C00824=1055.110,-115.851,435.627,170.509,28.358,155.374
C00825=1055.116,-115.601,435.618,170.511,28.358,155.374
C00826=1055.123,-115.318,435.607,170.513,28.359,155.373
C00827=1055.130,-115.034,435.597,170.515,28.360,155.373
C00828=1055.137,-114.749,435.585,170.517,28.360,155.373
C00829=1055.144,-114.466,435.574,170.520,28.361,155.373
C00830=1055.150,-114.216,435.565,170.522,28.362,155.373
C00831=1055.156,-113.966,435.555,170.524,28.362,155.373
C00832=1055.162,-113.716,435.546,170.526,28.363,155.373
C00833=1055.169,-113.466,435.536,170.528,28.364,155.373
C00834=1055.175,-113.217,435.526,170.530,28.364,155.373
C00835=1055.180,-112.966,435.516,170.532,28.365,155.373
C00836=1055.186,-112.717,435.507,170.534,28.366,155.373
C00837=1055.192,-112.467,435.497,170.536,28.367,155.373
C00838=1055.199,-112.217,435.488,170.538,28.367,155.373
C00839=1055.205,-111.968,435.477,170.540,28.368,155.373
C00840=1055.211,-111.718,435.468,170.542,28.369,155.373
C00841=1055.217,-111.468,435.458,170.544,28.369,155.373
C00842=1055.224,-111.219,435.449,170.547,28.370,155.373
C00843=1055.230,-110.969,435.439,170.548,28.371,155.373
C00844=1055.236,-110.719,435.429,170.550,28.372,155.373
C00845=1055.242,-110.470,435.419,170.552,28.372,155.372
C00846=1055.248,-110.220,435.409,170.554,28.373,155.372
C00847=1055.254,-109.970,435.399,170.556,28.374,155.372
C00848=1055.260,-109.720,435.390,170.558,28.374,155.372
C00849=1055.266,-109.470,435.380,170.561,28.375,155.372
C00850=1055.273,-109.221,435.370,170.562,28.376,155.372
C00851=1055.279,-108.971,435.360,170.564,28.376,155.372
C00852=1055.285,-108.721,435.351,170.566,28.377,155.372
C00853=1055.291,-108.472,435.341,170.568,28.378,155.372
C00854=1055.297,-108.222,435.331,170.570,28.379,155.372
C00855=1055.303,-107.972,435.321,170.572,28.379,155.372
C00856=1055.309,-107.723,435.311,170.575,28.381,155.372
C00857=1055.316,-107.473,435.302,170.577,28.381,155.372
C00858=1055.322,-107.224,435.291,170.578,28.382,155.372
C00859=1055.328,-106.974,435.282,170.580,28.383,155.372
C00860=1055.334,-106.724,435.272,170.582,28.384,155.372
C00861=1055.340,-106.474,435.262,170.584,28.384,155.372
C00862=1055.346,-106.225,435.252,170.586,28.385,155.372
C00863=1055.353,-105.975,435.242,170.589,28.386,155.372
C00864=1055.359,-105.724,435.232,170.591,28.387,155.372
C00865=1055.365,-105.475,435.221,170.592,28.388,155.372
C00866=1055.371,-105.225,435.212,170.594,28.388,155.372
C00867=1055.377,-104.975,435.202,170.596,28.389,155.372
C00868=1055.383,-104.726,435.191,170.598,28.390,155.372
C00869=1055.389,-104.476,435.182,170.600,28.391,155.372
C00870=1055.396,-104.227,435.172,170.602,28.392,155.372
C00871=1055.401,-103.977,435.161,170.605,28.393,155.372
C00872=1055.407,-103.727,435.152,170.606,28.394,155.372
C00873=1055.414,-103.478,435.142,170.608,28.394,155.371
C00874=1055.419,-103.228,435.131,170.610,28.395,155.372
C00875=1055.426,-102.978,435.121,170.612,28.396,155.372
C00876=1055.433,-102.728,435.111,170.614,28.397,155.371
C00877=1055.439,-102.478,435.102,170.616,28.398,155.371
C00878=1055.444,-102.229,435.091,170.617,28.399,155.372
C00879=1055.451,-101.979,435.081,170.620,28.400,155.371
C00880=1055.457,-101.730,435.071,170.622,28.401,155.371
C00881=1055.463,-101.480,435.061,170.624,28.402,155.371
C00882=1055.469,-101.230,435.051,170.626,28.402,155.371
C00883=1055.476,-100.980,435.041,170.628,28.403,155.371
C00884=1055.482,-100.730,435.030,170.630,28.404,155.371
C00885=1055.488,-100.481,435.020,170.631,28.405,155.371
C00886=1055.494,-100.232,435.010,170.633,28.406,155.371
C00887=1055.500,-99.981,435.000,170.636,28.407,155.371
C00888=1055.506,-99.732,434.989,170.638,28.408,155.371
C00889=1055.512,-99.481,434.979,170.640,28.409,155.371
C00890=1055.520,-99.197,434.968,170.642,28.410,155.371
C00891=1055.527,-98.911,434.956,170.644,28.411,155.371
C00892=1055.534,-98.625,434.944,170.646,28.412,155.371
C00893=1055.541,-98.340,434.932,170.649,28.413,155.371
C00894=1055.547,-98.090,434.922,170.651,28.414,155.371
C00895=1055.553,-97.840,434.912,170.653,28.415,155.371
C00896=1055.559,-97.591,434.902,170.655,28.416,155.371
C00897=1055.565,-97.340,434.891,170.656,28.417,155.371
C00898=1055.572,-97.091,434.881,170.658,28.418,155.371
C00899=1055.577,-96.841,434.870,170.660,28.419,155.371
C00900=1055.584,-96.592,434.860,170.662,28.420,155.371
C00901=1055.590,-96.343,434.849,170.665,28.421,155.371
C00902=1055.595,-96.092,434.839,170.666,28.422,155.371
C00903=1055.602,-95.843,434.828,170.668,28.423,155.371
C00904=1055.608,-95.593,434.818,170.670,28.424,155.372
C00905=1055.614,-95.343,434.808,170.672,28.425,155.372
C00906=1055.620,-95.094,434.797,170.674,28.426,155.371
C00907=1055.625,-94.844,434.786,170.676,28.427,155.371
C00908=1055.632,-94.594,434.776,170.677,28.428,155.372
C00909=1055.638,-94.344,434.765,170.679,28.429,155.372
C00910=1055.644,-94.095,434.755,170.682,28.430,155.372
C00911=1055.650,-93.845,434.745,170.684,28.431,155.372
C00912=1055.656,-93.595,434.734,170.686,28.432,155.372
C00913=1055.663,-93.346,434.723,170.688,28.433,155.372
C00914=1055.668,-93.096,434.713,170.689,28.435,155.372
C00915=1055.675,-92.846,434.703,170.691,28.436,155.372
C00916=1055.680,-92.597,434.692,170.693,28.437,155.372
C00917=1055.687,-92.347,434.681,170.695,28.438,155.372
C00918=1055.693,-92.097,434.671,170.698,28.439,155.372
C00919=1055.699,-91.847,434.660,170.699,28.440,155.372
C00920=1055.706,-91.597,434.650,170.701,28.441,155.372
C00921=1055.711,-91.348,434.639,170.703,28.442,155.372
C00922=1055.717,-91.099,434.628,170.705,28.443,155.372
C00923=1055.724,-90.849,434.618,170.707,28.445,155.372
C00924=1055.730,-90.599,434.607,170.709,28.446,155.372
C00925=1055.735,-90.349,434.596,170.710,28.447,155.372
C00926=1055.742,-90.100,434.586,170.712,28.448,155.372
C00927=1055.748,-89.850,434.575,170.715,28.449,155.372
C00928=1055.754,-89.600,434.564,170.717,28.450,155.372
C00929=1055.760,-89.351,434.554,170.719,28.451,155.372
C00930=1055.767,-89.101,434.542,170.720,28.452,155.372
C00931=1055.772,-88.851,434.532,170.722,28.453,155.372
C00932=1055.779,-88.602,434.522,170.724,28.454,155.372
C00933=1055.785,-88.351,434.511,170.726,28.456,155.372
C00934=1055.791,-88.102,434.500,170.728,28.457,155.372
C00935=1055.797,-87.853,434.490,170.730,28.458,155.372
C00936=1055.804,-87.602,434.478,170.731,28.459,155.372
C00937=1055.809,-87.353,434.467,170.734,28.461,155.372
C00938=1055.816,-87.104,434.457,170.736,28.462,155.373
C00939=1055.822,-86.854,434.446,170.738,28.463,155.373
C00940=1055.828,-86.604,434.435,170.740,28.464,155.373
C00941=1055.834,-86.355,434.425,170.741,28.465,155.373
C00942=1055.841,-86.105,434.413,170.743,28.466,155.373
C00943=1055.846,-85.855,434.403,170.745,28.467,155.373
C00944=1055.853,-85.605,434.393,170.747,28.469,155.373
C00945=1055.859,-85.355,434.382,170.749,28.470,155.373
C00946=1055.865,-85.106,434.371,170.751,28.471,155.373
C00947=1055.872,-84.856,434.360,170.753,28.472,155.373
C00948=1055.878,-84.606,434.349,170.755,28.473,155.373
C00949=1055.884,-84.356,434.338,170.757,28.474,155.373
C00950=1055.890,-84.107,434.328,170.759,28.476,155.373
C00951=1055.896,-83.858,434.316,170.761,28.477,155.373
C00952=1055.903,-83.608,434.305,170.762,28.478,155.373
C00953=1055.908,-83.358,434.294,170.764,28.479,155.373
C00954=1055.916,-83.075,434.282,170.767,28.480,155.373
C00955=1055.923,-82.791,434.270,170.769,28.482,155.373
C00956=1055.930,-82.508,434.258,170.771,28.483,155.373
C00957=1055.937,-82.225,434.245,170.773,28.485,155.373
C00958=1055.943,-81.976,434.234,170.775,28.486,155.373
C00959=1055.950,-81.726,434.223,170.777,28.487,155.373
C00960=1055.956,-81.476,434.212,170.779,28.488,155.374
C00961=1055.962,-81.226,434.201,170.781,28.489,155.374
C00962=1055.968,-80.977,434.190,170.782,28.491,155.374
C00963=1055.975,-80.727,434.180,170.784,28.492,155.374
C00964=1055.981,-80.478,434.168,170.787,28.493,155.374
C00965=1055.987,-80.228,434.157,170.789,28.494,155.374
C00966=1055.993,-79.978,434.146,170.790,28.496,155.374
C00967=1056.000,-79.728,434.135,170.792,28.497,155.374
C00968=1056.006,-79.479,434.124,170.794,28.498,155.374
C00969=1056.012,-79.229,434.113,170.796,28.499,155.374
C00970=1056.018,-78.980,434.102,170.798,28.500,155.374
C00971=1056.025,-78.730,434.090,170.799,28.502,155.374
C00972=1056.030,-78.480,434.079,170.801,28.503,155.374
C00973=1056.037,-78.230,434.068,170.803,28.504,155.374
C00974=1056.042,-77.980,434.057,170.805,28.506,155.374
C00975=1056.049,-77.731,434.045,170.808,28.507,155.374
C00976=1056.055,-77.481,434.034,170.809,28.509,155.375
C00977=1056.061,-77.231,434.023,170.811,28.510,155.375
C00978=1056.067,-76.982,434.012,170.813,28.511,155.375
C00979=1056.073,-76.732,434.000,170.815,28.512,155.375
C00980=1056.079,-76.483,433.989,170.817,28.513,155.375
C00981=1056.086,-76.232,433.978,170.818,28.515,155.375
C00982=1056.092,-75.983,433.967,170.820,28.516,155.375
C00983=1056.098,-75.733,433.955,170.822,28.518,155.375
C00984=1056.104,-75.484,433.945,170.824,28.519,155.375
C00985=1056.110,-75.234,433.933,170.826,28.520,155.375
C00986=1056.116,-74.985,433.922,170.827,28.522,155.375
C00987=1056.122,-74.735,433.910,170.830,28.523,155.376
C00988=1056.128,-74.485,433.900,170.832,28.524,155.376
C00989=1056.135,-74.235,433.888,170.834,28.526,155.376
C00990=1056.141,-73.986,433.877,170.836,28.527,155.376
C00991=1056.147,-73.736,433.865,170.837,28.529,155.376
C00992=1056.153,-73.487,433.854,170.839,28.530,155.376
C00993=1056.159,-73.237,433.843,170.841,28.531,155.376
C00994=1056.166,-72.987,433.831,170.843,28.533,155.376
C00995=1056.171,-72.737,433.819,170.844,28.534,155.376
C00996=1056.177,-72.487,433.808,170.846,28.536,155.376
C00997=1056.183,-72.238,433.796,170.848,28.537,155.377
C00998=1056.190,-71.988,433.785,170.850,28.539,155.377
C00999=1056.196,-71.739,433.774,170.852,28.540,155.377
C01000=1056.201,-71.489,433.762,170.853,28.542,155.377
C01001=1056.207,-71.240,433.750,170.856,28.543,155.377
C01002=1056.214,-70.990,433.739,170.858,28.545,155.377
C01003=1056.220,-70.741,433.727,170.860,28.546,155.377
C01004=1056.225,-70.490,433.715,170.861,28.548,155.377
C01005=1056.231,-70.241,433.704,170.863,28.549,155.377
C01006=1056.238,-69.991,433.693,170.865,28.551,155.377
C01007=1056.244,-69.742,433.681,170.867,28.552,155.378
C01008=1056.249,-69.492,433.669,170.868,28.553,155.378
C01009=1056.256,-69.242,433.657,170.870,28.555,155.378
C01010=1056.262,-68.993,433.646,170.872,28.557,155.378
C01011=1056.268,-68.743,433.634,170.874,28.558,155.378
C01012=1056.273,-68.493,433.623,170.876,28.559,155.378
C01013=1056.280,-68.244,433.611,170.877,28.561,155.378
C01014=1056.286,-67.994,433.600,170.879,28.563,155.378
C01015=1056.292,-67.745,433.588,170.881,28.564,155.379
C01016=1056.298,-67.495,433.576,170.883,28.565,155.379
C01017=1056.305,-67.245,433.564,170.885,28.567,155.379
C01018=1056.312,-66.964,433.552,170.887,28.569,155.379
C01019=1056.318,-66.682,433.538,170.889,28.571,155.379
C01020=1056.326,-66.402,433.525,170.891,28.572,155.379
C01021=1056.332,-66.121,433.511,170.893,28.574,155.379
C01022=1056.338,-65.871,433.501,170.895,28.576,155.379
C01023=1056.345,-65.622,433.489,170.897,28.577,155.380
C01024=1056.351,-65.372,433.476,170.899,28.578,155.380
C01025=1056.356,-65.122,433.465,170.900,28.580,155.380
C01026=1056.363,-64.873,433.453,170.902,28.582,155.380
C01027=1056.369,-64.623,433.441,170.904,28.583,155.380
C01028=1056.375,-64.373,433.430,170.906,28.584,155.380
C01029=1056.381,-64.124,433.418,170.908,28.586,155.380
C01030=1056.387,-63.874,433.405,170.909,28.588,155.380
C01031=1056.393,-63.624,433.394,170.911,28.589,155.381
C01032=1056.400,-63.375,433.382,170.913,28.591,155.381
C01033=1056.406,-63.125,433.370,170.915,28.593,155.381
C01034=1056.411,-62.876,433.358,170.917,28.594,155.381
C01035=1056.418,-62.626,433.347,170.919,28.595,155.381
C01036=1056.424,-62.376,433.335,170.921,28.597,155.381
C01037=1056.430,-62.126,433.322,170.923,28.599,155.381
C01038=1056.436,-61.877,433.311,170.924,28.600,155.381
C01039=1056.443,-61.627,433.300,170.926,28.602,155.382
C01040=1056.449,-61.377,433.287,170.928,28.603,155.382
C01041=1056.455,-61.128,433.275,170.930,28.605,155.382
C01042=1056.461,-60.879,433.264,170.931,28.606,155.382
C01043=1056.467,-60.628,433.252,170.933,28.608,155.382
C01044=1056.474,-60.379,433.240,170.935,28.610,155.382
C01045=1056.480,-60.129,433.228,170.937,28.611,155.382
C01046=1056.486,-59.880,433.216,170.938,28.613,155.382
C01047=1056.492,-59.631,433.204,170.940,28.614,155.382
C01048=1056.499,-59.381,433.192,170.942,28.616,155.383
C01049=1056.504,-59.130,433.180,170.944,28.617,155.383
C01050=1056.511,-58.882,433.168,170.946,28.619,155.383
C01051=1056.516,-58.632,433.156,170.947,28.621,155.383
C01052=1056.523,-58.382,433.144,170.949,28.622,155.383
C01053=1056.530,-58.133,433.132,170.951,28.624,155.383
C01054=1056.536,-57.883,433.119,170.953,28.625,155.384
C01055=1056.542,-57.633,433.107,170.954,28.627,155.384
C01056=1056.548,-57.384,433.096,170.957,28.628,155.384
C01057=1056.554,-57.134,433.084,170.959,28.630,155.384
C01058=1056.561,-56.884,433.072,170.961,28.632,155.384
C01059=1056.567,-56.635,433.060,170.962,28.633,155.384
C01060=1056.573,-56.385,433.047,170.964,28.635,155.384
C01061=1056.580,-56.135,433.035,170.966,28.637,155.384
C01062=1056.585,-55.886,433.023,170.968,28.638,155.385
C01063=1056.592,-55.636,433.011,170.969,28.640,155.385
C01064=1056.598,-55.387,432.999,170.971,28.642,155.385
C01065=1056.604,-55.137,432.987,170.973,28.643,155.385
C01066=1056.611,-54.887,432.975,170.975,28.645,155.385
C01067=1056.617,-54.637,432.962,170.976,28.646,155.385
C01068=1056.623,-54.388,432.950,170.978,28.648,155.385
C01069=1056.630,-54.138,432.938,170.980,28.650,155.386
C01070=1056.635,-53.889,432.926,170.982,28.651,155.386
C01071=1056.642,-53.640,432.914,170.983,28.653,155.386
C01072=1056.648,-53.390,432.902,170.985,28.655,155.386
C01073=1056.655,-53.140,432.890,170.987,28.656,155.386
C01074=1056.661,-52.891,432.878,170.989,28.657,155.386
C01075=1056.667,-52.641,432.865,170.991,28.659,155.386
C01076=1056.674,-52.391,432.853,170.992,28.661,155.387
C01077=1056.680,-52.141,432.841,170.994,28.662,155.387
C01078=1056.686,-51.892,432.829,170.996,28.664,155.387
C01079=1056.692,-51.642,432.816,170.998,28.665,155.387
C01080=1056.699,-51.392,432.804,170.999,28.667,155.387
C01081=1056.706,-51.143,432.792,171.001,28.669,155.387
C01082=1056.712,-50.863,432.778,171.004,28.671,155.388
C01083=1056.719,-50.584,432.765,171.006,28.673,155.388
C01084=1056.727,-50.304,432.750,171.007,28.674,155.388
C01085=1056.733,-50.024,432.737,171.009,28.677,155.388
C01086=1056.739,-49.774,432.724,171.011,28.678,155.388
C01087=1056.746,-49.525,432.712,171.012,28.680,155.388
C01088=1056.752,-49.275,432.699,171.014,28.682,155.389
C01089=1056.758,-49.025,432.686,171.017,28.683,155.389
C01090=1056.763,-48.775,432.674,171.019,28.686,155.389
C01091=1056.770,-48.526,432.662,171.020,28.687,155.389
C01092=1056.776,-48.277,432.649,171.022,28.689,155.389
C01093=1056.782,-48.027,432.636,171.024,28.691,155.389
C01094=1056.788,-47.777,432.624,171.026,28.693,155.390
C01095=1056.794,-47.528,432.612,171.027,28.695,155.390
C01096=1056.800,-47.278,432.599,171.029,28.696,155.390
C01097=1056.806,-47.029,432.586,171.031,28.698,155.390
C01098=1056.813,-46.779,432.574,171.033,28.700,155.390
C01099=1056.819,-46.529,432.562,171.034,28.702,155.390
C01100=1056.825,-46.279,432.549,171.036,28.703,155.391
C01101=1056.831,-46.030,432.536,171.038,28.705,155.391
C01102=1056.837,-45.780,432.523,171.040,28.707,155.391
C01103=1056.844,-45.531,432.511,171.041,28.709,155.391
C01104=1056.850,-45.281,432.498,171.043,28.710,155.391
C01105=1056.856,-45.031,432.485,171.045,28.712,155.392
C01106=1056.862,-44.782,432.473,171.047,28.714,155.392
C01107=1056.869,-44.533,432.460,171.048,28.716,155.392
C01108=1056.874,-44.283,432.448,171.050,28.718,155.392
C01109=1056.880,-44.033,432.435,171.052,28.720,155.392
C01110=1056.887,-43.784,432.422,171.053,28.721,155.392
C01111=1056.892,-43.534,432.409,171.055,28.723,155.393
C01112=1056.899,-43.284,432.397,171.057,28.725,155.393
C01113=1056.905,-43.035,432.384,171.059,28.727,155.393
C01114=1056.911,-42.785,432.372,171.060,28.729,155.393
C01115=1056.917,-42.535,432.359,171.062,28.730,155.393
C01116=1056.924,-42.286,432.346,171.064,28.732,155.394
C01117=1056.930,-42.036,432.334,171.066,28.734,155.394
C01118=1056.936,-41.787,432.320,171.067,28.736,155.394
C01119=1056.942,-41.537,432.308,171.069,28.737,155.394
C01120=1056.948,-41.287,432.295,171.071,28.740,155.394
C01121=1056.954,-41.038,432.282,171.072,28.741,155.395
C01122=1056.961,-40.788,432.270,171.073,28.743,155.395
C01123=1056.967,-40.539,432.257,171.075,28.745,155.395
C01124=1056.973,-40.289,432.244,171.077,28.746,155.395
C01125=1056.979,-40.040,432.231,171.079,28.748,155.395
C01126=1056.985,-39.790,432.219,171.080,28.750,155.396
C01127=1056.992,-39.541,432.206,171.082,28.752,155.396
C01128=1056.998,-39.291,432.193,171.084,28.754,155.396
C01129=1057.005,-39.041,432.180,171.086,28.756,155.396
C01130=1057.011,-38.791,432.167,171.087,28.757,155.396
C01131=1057.017,-38.542,432.154,171.089,28.760,155.397
C01132=1057.023,-38.292,432.141,171.091,28.761,155.397
C01133=1057.029,-38.043,432.128,171.093,28.763,155.397
C01134=1057.035,-37.793,432.115,171.094,28.765,155.397
C01135=1057.041,-37.544,432.102,171.096,28.767,155.397
C01136=1057.047,-37.294,432.090,171.098,28.769,155.398
C01137=1057.053,-37.045,432.076,171.099,28.771,155.398
C01138=1057.059,-36.795,432.064,171.101,28.773,155.398
C01139=1057.065,-36.546,432.051,171.103,28.774,155.398
C01140=1057.072,-36.296,432.037,171.105,28.777,155.398
C01141=1057.078,-36.046,432.025,171.106,28.778,155.398
C01142=1057.084,-35.796,432.011,171.108,28.781,155.399
C01143=1057.090,-35.547,431.999,171.110,28.782,155.399
C01144=1057.097,-35.297,431.985,171.111,28.784,155.399
C01145=1057.103,-35.048,431.972,171.113,28.786,155.399
C01146=1057.109,-34.769,431.958,171.115,28.788,155.400
C01147=1057.116,-34.489,431.943,171.117,28.791,155.400
C01148=1057.123,-34.210,431.928,171.119,28.793,155.400
C01149=1057.130,-33.931,431.913,171.121,28.795,155.400
C01150=1057.136,-33.681,431.900,171.123,28.797,155.401
C01151=1057.142,-33.431,431.887,171.124,28.799,155.401
C01152=1057.148,-33.181,431.874,171.126,28.801,155.401
C01153=1057.155,-32.932,431.861,171.128,28.803,155.401
C01154=1057.161,-32.682,431.848,171.130,28.805,155.401
C01155=1057.167,-32.433,431.835,171.131,28.807,155.402
C01156=1057.173,-32.184,431.821,171.133,28.808,155.402
C01157=1057.179,-31.934,431.808,171.134,28.810,155.402
C01158=1057.186,-31.684,431.795,171.136,28.813,155.402
C01159=1057.191,-31.434,431.781,171.137,28.814,155.402
C01160=1057.197,-31.185,431.768,171.139,28.816,155.403
C01161=1057.204,-30.936,431.755,171.141,28.818,155.403
C01162=1057.210,-30.686,431.742,171.142,28.820,155.403
C01163=1057.216,-30.437,431.729,171.144,28.822,155.403
C01164=1057.223,-30.187,431.715,171.146,28.824,155.404
C01165=1057.229,-29.937,431.702,171.148,28.826,155.404
C01166=1057.235,-29.688,431.689,171.149,28.828,155.404
C01167=1057.241,-29.438,431.676,171.151,28.830,155.404
C01168=1057.248,-29.188,431.663,171.153,28.832,155.404
C01169=1057.253,-28.939,431.649,171.155,28.834,155.405
C01170=1057.259,-28.689,431.636,171.156,28.836,155.405
C01171=1057.266,-28.440,431.622,171.158,28.838,155.405
C01172=1057.272,-28.191,431.609,171.160,28.840,155.405
C01173=1057.278,-27.940,431.596,171.161,28.842,155.406
C01174=1057.285,-27.691,431.583,171.163,28.844,155.406
C01175=1057.291,-27.442,431.570,171.165,28.846,155.406
C01176=1057.298,-27.192,431.556,171.167,28.848,155.406
C01177=1057.303,-26.942,431.542,171.168,28.849,155.406
C01178=1057.309,-26.693,431.529,171.169,28.851,155.407
C01179=1057.315,-26.444,431.515,171.171,28.854,155.407
C01180=1057.322,-26.194,431.502,171.173,28.855,155.407
C01181=1057.327,-25.944,431.489,171.174,28.858,155.407
C01182=1057.334,-25.694,431.475,171.176,28.860,155.408
C01183=1057.340,-25.445,431.462,171.178,28.862,155.408
C01184=1057.345,-25.195,431.448,171.179,28.864,155.408
C01185=1057.352,-24.946,431.435,171.181,28.866,155.408
C01186=1057.358,-24.696,431.421,171.183,28.868,155.409
C01187=1057.364,-24.447,431.408,171.185,28.870,155.409
C01188=1057.370,-24.197,431.394,171.186,28.872,155.409
C01189=1057.376,-23.947,431.380,171.188,28.874,155.409
C01190=1057.382,-23.698,431.367,171.190,28.876,155.410
C01191=1057.389,-23.449,431.353,171.191,28.879,155.410
C01192=1057.395,-23.198,431.339,171.193,28.880,155.410
C01193=1057.401,-22.949,431.326,171.194,28.882,155.410
C01194=1057.407,-22.700,431.313,171.196,28.884,155.411
C01195=1057.413,-22.450,431.299,171.197,28.887,155.411
C01196=1057.419,-22.200,431.285,171.199,28.888,155.411
C01197=1057.426,-21.952,431.271,171.201,28.890,155.411
C01198=1057.431,-21.702,431.257,171.202,28.893,155.412
C01199=1057.438,-21.452,431.244,171.204,28.895,155.412
C01200=1057.444,-21.203,431.230,171.206,28.896,155.412
C01201=1057.450,-20.953,431.217,171.208,28.899,155.412
C01202=1057.457,-20.703,431.203,171.209,28.901,155.412
C01203=1057.462,-20.454,431.189,171.211,28.903,155.413
C01204=1057.468,-20.204,431.176,171.213,28.905,155.413
C01205=1057.474,-19.954,431.162,171.214,28.907,155.413
C01206=1057.481,-19.705,431.148,171.215,28.909,155.413
C01207=1057.487,-19.456,431.134,171.217,28.911,155.414
C01208=1057.493,-19.206,431.120,171.219,28.913,155.414
C01209=1057.500,-18.957,431.107,171.220,28.915,155.414
C01210=1057.506,-18.676,431.091,171.222,28.918,155.415
C01211=1057.513,-18.397,431.076,171.225,28.920,155.415
C01212=1057.520,-18.116,431.060,171.226,28.922,155.415
C01213=1057.528,-17.836,431.045,171.228,28.925,155.415
C01214=1057.533,-17.587,431.031,171.230,28.927,155.416
C01215=1057.540,-17.337,431.017,171.231,28.929,155.416
C01216=1057.546,-17.088,431.004,171.233,28.931,155.416
C01217=1057.551,-16.838,430.990,171.235,28.933,155.416
C01218=1057.559,-16.589,430.976,171.236,28.935,155.417
C01219=1057.564,-16.339,430.962,171.237,28.937,155.417
C01220=1057.571,-16.089,430.948,171.239,28.939,155.417
C01221=1057.576,-15.839,430.934,171.241,28.941,155.417
C01222=1057.583,-15.591,430.920,171.243,28.943,155.418
C01223=1057.590,-15.341,430.907,171.244,28.945,155.418
C01224=1057.595,-15.091,430.893,171.246,28.948,155.418
C01225=1057.602,-14.841,430.879,171.248,28.950,155.418
C01226=1057.608,-14.592,430.865,171.249,28.952,155.419
C01227=1057.613,-14.343,430.851,171.251,28.954,155.419
C01228=1057.620,-14.093,430.837,171.252,28.956,155.419
C01229=1057.626,-13.844,430.823,171.254,28.958,155.419
C01230=1057.632,-13.594,430.808,171.255,28.960,155.420
C01231=1057.638,-13.344,430.795,171.257,28.962,155.420
C01232=1057.644,-13.095,430.781,171.259,28.965,155.420
C01233=1057.650,-12.845,430.766,171.260,28.967,155.420
C01234=1057.656,-12.596,430.753,171.262,28.969,155.421
C01235=1057.663,-12.346,430.738,171.264,28.971,155.421
C01236=1057.668,-12.097,430.724,171.266,28.973,155.421
C01237=1057.675,-11.847,430.710,171.267,28.976,155.422
C01238=1057.681,-11.598,430.696,171.268,28.978,155.422
C01239=1057.686,-11.348,430.682,171.270,28.980,155.422
C01240=1057.693,-11.099,430.668,171.271,28.982,155.422
C01241=1057.699,-10.849,430.654,171.273,28.984,155.423
C01242=1057.706,-10.600,430.640,171.275,28.986,155.423
C01243=1057.711,-10.350,430.626,171.277,28.989,155.423
C01244=1057.718,-10.101,430.611,171.278,28.991,155.423
C01245=1057.723,-9.851,430.597,171.280,28.993,155.424
C01246=1057.730,-9.601,430.583,171.282,28.995,155.424
C01247=1057.736,-9.352,430.569,171.282,28.997,155.424
C01248=1057.742,-9.102,430.554,171.284,28.999,155.425
C01249=1057.748,-8.853,430.540,171.286,29.002,155.425
C01250=1057.754,-8.603,430.526,171.287,29.004,155.425
C01251=1057.760,-8.354,430.512,171.289,29.006,155.425
C01252=1057.767,-8.104,430.498,171.291,29.008,155.426
C01253=1057.773,-7.855,430.483,171.293,29.010,155.426
C01254=1057.779,-7.605,430.469,171.294,29.013,155.426
C01255=1057.785,-7.356,430.455,171.296,29.015,155.426
C01256=1057.792,-7.106,430.440,171.297,29.017,155.427
C01257=1057.797,-6.857,430.426,171.298,29.019,155.427
C01258=1057.804,-6.607,430.411,171.300,29.021,155.427
C01259=1057.810,-6.358,430.398,171.302,29.024,155.428
C01260=1057.816,-6.108,430.383,171.304,29.026,155.428
C01261=1057.822,-5.858,430.369,171.305,29.028,155.428
C01262=1057.832,-5.474,430.347,171.308,29.031,155.429
C01263=1057.841,-5.089,430.325,171.310,29.035,155.429
C01264=1057.851,-4.705,430.303,171.312,29.037,155.429
C01265=1057.861,-4.320,430.281,171.315,29.041,155.430
C01266=1057.867,-4.071,430.267,171.316,29.043,155.430
C01267=1057.873,-3.821,430.252,171.318,29.045,155.430
C01268=1057.879,-3.572,430.238,171.320,29.048,155.431
C01269=1057.885,-3.322,430.223,171.321,29.050,155.431
C01270=1057.895,-2.927,430.200,171.324,29.053,155.431
C01271=1057.904,-2.530,430.178,171.327,29.057,155.432
C01272=1057.914,-2.133,430.154,171.329,29.061,155.432
C01273=1057.924,-1.737,430.131,171.332,29.064,155.433
C01274=1057.929,-1.488,430.116,171.333,29.066,155.433
C01275=1057.936,-1.239,430.101,171.334,29.069,155.433
C01276=1057.942,-0.988,430.087,171.336,29.071,155.434
C01277=1057.948,-0.739,430.072,171.337,29.073,155.434
C01278=1057.954,-0.490,430.057,171.339,29.076,155.434
C01279=1057.960,-0.241,430.043,171.341,29.078,155.435
C01280=1057.966,0.009,430.029,171.343,29.080,155.435
C01281=1057.972,0.258,430.014,171.343,29.083,155.435
C01282=1057.978,0.508,429.999,171.345,29.085,155.436
C01283=1057.984,0.758,429.984,171.347,29.087,155.436
C01284=1057.990,1.007,429.970,171.348,29.089,155.436
C01285=1057.997,1.256,429.955,171.350,29.091,155.436
C01286=1058.002,1.506,429.941,171.352,29.094,155.437
C01287=1058.008,1.756,429.926,171.353,29.096,155.437
C01288=1058.015,2.005,429.911,171.354,29.098,155.437
C01289=1058.021,2.254,429.896,171.356,29.101,155.438
C01290=1058.027,2.504,429.881,171.358,29.103,155.438
C01291=1058.033,2.753,429.867,171.359,29.106,155.438
C01292=1058.039,3.003,429.852,171.361,29.108,155.439
C01293=1058.045,3.253,429.838,171.363,29.110,155.439
C01294=1058.051,3.502,429.823,171.364,29.112,155.439
C01295=1058.057,3.751,429.808,171.365,29.114,155.439
C01296=1058.064,4.001,429.793,171.367,29.117,155.440
C01297=1058.070,4.250,429.778,171.368,29.119,155.440
C01298=1058.075,4.500,429.763,171.370,29.121,155.440
C01299=1058.082,4.750,429.748,171.372,29.124,155.441
C01300=1058.087,4.999,429.733,171.374,29.126,155.441
C01301=1058.094,5.248,429.718,171.374,29.128,155.441
C01302=1058.100,5.498,429.704,171.376,29.131,155.442
C01303=1058.106,5.747,429.689,171.378,29.133,155.442
C01304=1058.112,5.996,429.674,171.379,29.135,155.442
C01305=1058.119,6.246,429.659,171.381,29.137,155.442
C01306=1058.125,6.495,429.644,171.383,29.140,155.443
C01307=1058.131,6.745,429.630,171.384,29.142,155.443
C01308=1058.137,6.994,429.615,171.385,29.144,155.443
C01309=1058.144,7.244,429.600,171.387,29.146,155.444
C01310=1058.149,7.493,429.585,171.389,29.148,155.444
C01311=1058.155,7.743,429.570,171.390,29.151,155.444
C01312=1058.161,7.993,429.555,171.392,29.153,155.445
C01313=1058.168,8.242,429.540,171.394,29.156,155.445
C01314=1058.174,8.491,429.525,171.395,29.158,155.445
C01315=1058.180,8.741,429.510,171.396,29.160,155.445
C01316=1058.186,8.991,429.495,171.398,29.163,155.446
C01317=1058.193,9.240,429.480,171.400,29.165,155.446
C01318=1058.199,9.489,429.466,171.401,29.167,155.446
C01319=1058.205,9.739,429.451,171.403,29.169,155.447
C01320=1058.211,9.988,429.436,171.404,29.171,155.447
C01321=1058.217,10.238,429.420,171.406,29.174,155.447
C01322=1058.223,10.487,429.406,171.407,29.176,155.448
C01323=1058.229,10.737,429.391,171.409,29.178,155.448
C01324=1058.236,10.987,429.376,171.411,29.181,155.448
C01325=1058.242,11.236,429.360,171.412,29.183,155.449
C01326=1058.249,11.485,429.345,171.413,29.185,155.449
C01327=1058.254,11.734,429.331,171.415,29.188,155.449
C01328=1058.261,11.984,429.316,171.417,29.190,155.449
C01329=1058.266,12.234,429.300,171.418,29.192,155.450
C01330=1058.273,12.484,429.285,171.420,29.195,155.450
C01331=1058.279,12.733,429.269,171.422,29.197,155.450
C01332=1058.285,12.982,429.255,171.422,29.199,155.451
C01333=1058.292,13.231,429.240,171.424,29.201,155.451
C01334=1058.299,13.516,429.223,171.426,29.204,155.451
C01335=1058.306,13.799,429.206,171.427,29.207,155.452
C01336=1058.313,14.083,429.188,171.429,29.209,155.452
C01337=1058.320,14.366,429.171,171.431,29.212,155.452
C01338=1058.326,14.616,429.156,171.432,29.214,155.453
C01339=1058.332,14.866,429.141,171.434,29.217,155.453
C01340=1058.338,15.114,429.125,171.436,29.219,155.453
C01341=1058.344,15.364,429.110,171.438,29.221,155.454
C01342=1058.350,15.614,429.095,171.439,29.224,155.454
C01343=1058.357,15.863,429.079,171.440,29.226,155.454
C01344=1058.363,16.113,429.064,171.442,29.228,155.455
C01345=1058.369,16.362,429.049,171.443,29.231,155.455
C01346=1058.374,16.611,429.034,171.445,29.233,155.455
C01347=1058.381,16.861,429.018,171.447,29.235,155.455
C01348=1058.387,17.110,429.003,171.448,29.238,155.456
C01349=1058.393,17.360,428.987,171.449,29.240,155.456
C01350=1058.400,17.609,428.972,171.451,29.242,155.456
C01351=1058.406,17.859,428.957,171.453,29.245,155.457
C01352=1058.411,18.108,428.942,171.454,29.247,155.457
C01353=1058.418,18.357,428.926,171.456,29.249,155.457
C01354=1058.423,18.607,428.910,171.457,29.252,155.458
C01355=1058.430,18.856,428.895,171.458,29.254,155.458
C01356=1058.436,19.106,428.880,171.460,29.256,155.458
C01357=1058.442,19.356,428.864,171.462,29.259,155.459
C01358=1058.449,19.605,428.849,171.464,29.261,155.459
C01359=1058.454,19.855,428.833,171.464,29.264,155.459
C01360=1058.461,20.103,428.818,171.466,29.266,155.460
C01361=1058.467,20.353,428.803,171.468,29.268,155.460
C01362=1058.473,20.602,428.787,171.469,29.271,155.460
C01363=1058.479,20.852,428.772,171.471,29.273,155.461
C01364=1058.485,21.102,428.756,171.472,29.276,155.461
C01365=1058.492,21.351,428.740,171.474,29.278,155.461
C01366=1058.497,21.601,428.725,171.475,29.280,155.462
C01367=1058.503,21.850,428.709,171.477,29.283,155.462
C01368=1058.510,22.100,428.694,171.479,29.285,155.462
C01369=1058.515,22.348,428.678,171.479,29.288,155.463
C01370=1058.521,22.598,428.663,171.481,29.290,155.463
C01371=1058.527,22.847,428.647,171.483,29.292,155.463
C01372=1058.534,23.097,428.632,171.484,29.295,155.464
C01373=1058.540,23.346,428.615,171.486,29.297,155.464
C01374=1058.546,23.596,428.600,171.487,29.299,155.464
C01375=1058.552,23.845,428.584,171.489,29.302,155.465
C01376=1058.559,24.094,428.569,171.490,29.304,155.465
C01377=1058.564,24.344,428.553,171.492,29.307,155.465
C01378=1058.571,24.593,428.537,171.494,29.309,155.466
C01379=1058.577,24.843,428.522,171.494,29.311,155.466
C01380=1058.583,25.092,428.506,171.496,29.314,155.466
C01381=1058.589,25.342,428.491,171.498,29.316,155.467
C01382=1058.595,25.592,428.474,171.500,29.318,155.467
C01383=1058.602,25.841,428.459,171.501,29.321,155.467
C01384=1058.607,26.091,428.443,171.502,29.323,155.468
C01385=1058.613,26.339,428.428,171.504,29.325,155.468
C01386=1058.619,26.589,428.412,171.505,29.328,155.468
C01387=1058.626,26.838,428.397,171.507,29.330,155.469
C01388=1058.632,27.087,428.380,171.509,29.333,155.469
C01389=1058.637,27.337,428.365,171.510,29.335,155.469
C01390=1058.644,27.586,428.349,171.511,29.337,155.470
C01391=1058.650,27.836,428.333,171.513,29.340,155.470
C01392=1058.656,28.086,428.318,171.515,29.342,155.470
C01393=1058.662,28.335,428.302,171.516,29.345,155.471
C01394=1058.668,28.584,428.285,171.517,29.347,155.471
C01395=1058.675,28.833,428.270,171.519,29.350,155.471
C01396=1058.680,29.083,428.254,171.521,29.352,155.472
C01397=1058.686,29.333,428.238,171.522,29.355,155.472
C01398=1058.693,29.618,428.220,171.524,29.357,155.472
C01399=1058.701,29.903,428.201,171.526,29.360,155.473
C01400=1058.707,30.187,428.183,171.527,29.363,155.473
C01401=1058.714,30.473,428.165,171.529,29.366,155.474
C01402=1058.721,30.722,428.149,171.531,29.368,155.474
C01403=1058.727,30.971,428.133,171.531,29.371,155.474
C01404=1058.733,31.221,428.117,171.533,29.373,155.475
C01405=1058.738,31.471,428.101,171.535,29.375,155.475
C01406=1058.744,31.720,428.085,171.536,29.378,155.475
C01407=1058.751,31.969,428.070,171.538,29.380,155.476
C01408=1058.757,32.218,428.053,171.539,29.382,155.476
C01409=1058.763,32.468,428.037,171.541,29.385,155.476
C01410=1058.768,32.718,428.021,171.542,29.387,155.477
C01411=1058.775,32.967,428.006,171.544,29.390,155.477
C01412=1058.781,33.216,427.990,171.546,29.392,155.477
C01413=1058.787,33.466,427.973,171.546,29.395,155.478
C01414=1058.793,33.715,427.957,171.548,29.397,155.478
C01415=1058.799,33.964,427.941,171.550,29.400,155.478
C01416=1058.806,34.214,427.925,171.552,29.402,155.479
C01417=1058.812,34.463,427.908,171.552,29.405,155.479
C01418=1058.818,34.713,427.893,171.554,29.407,155.479
C01419=1058.824,34.963,427.877,171.556,29.410,155.480
C01420=1058.830,35.212,427.860,171.557,29.412,155.480
C01421=1058.836,35.461,427.845,171.559,29.414,155.480
C01422=1058.842,35.710,427.829,171.560,29.416,155.481
C01423=1058.848,35.960,427.812,171.562,29.419,155.481
C01424=1058.854,36.209,427.796,171.563,29.422,155.482
C01425=1058.860,36.458,427.780,171.565,29.424,155.482
C01426=1058.867,36.707,427.764,171.566,29.427,155.482
C01427=1058.873,36.957,427.747,171.567,29.429,155.483
C01428=1058.879,37.207,427.731,171.569,29.432,155.483
C01429=1058.885,37.456,427.715,171.571,29.434,155.483
C01430=1058.891,37.706,427.699,171.572,29.437,155.484
C01431=1058.897,37.955,427.682,171.573,29.439,155.484
C01432=1058.903,38.204,427.666,171.575,29.441,155.484
C01433=1058.909,38.454,427.650,171.577,29.443,155.485
C01434=1058.915,38.703,427.634,171.578,29.446,155.485
C01435=1058.921,38.952,427.617,171.579,29.449,155.485
C01436=1058.928,39.202,427.601,171.581,29.451,155.486
C01437=1058.934,39.452,427.585,171.582,29.454,155.486
C01438=1058.940,39.701,427.568,171.584,29.456,155.486
C01439=1058.945,39.950,427.552,171.586,29.459,155.487
C01440=1058.951,40.200,427.536,171.587,29.461,155.487
C01441=1058.957,40.449,427.519,171.588,29.463,155.487
C01442=1058.963,40.698,427.503,171.590,29.466,155.488
C01443=1058.970,40.947,427.486,171.592,29.468,155.488
C01444=1058.976,41.197,427.470,171.592,29.471,155.489
C01445=1058.982,41.447,427.453,171.594,29.474,155.489
C01446=1058.988,41.696,427.437,171.596,29.476,155.489
C01447=1058.994,41.945,427.421,171.598,29.479,155.490
C01448=1059.000,42.195,427.405,171.599,29.481,155.490
C01449=1059.006,42.444,427.388,171.600,29.483,155.490
C01450=1059.012,42.694,427.372,171.602,29.486,155.491
C01451=1059.019,42.943,427.355,171.603,29.488,155.491
C01452=1059.025,43.192,427.339,171.605,29.491,155.491
C01453=1059.031,43.441,427.322,171.606,29.493,155.492
C01454=1059.037,43.691,427.306,171.608,29.496,155.492
C01455=1059.043,43.940,427.290,171.609,29.499,155.493
C01456=1059.049,44.190,427.272,171.611,29.501,155.493
C01457=1059.055,44.439,427.256,171.612,29.503,155.493
C01458=1059.061,44.689,427.239,171.613,29.506,155.494
C01459=1059.066,44.938,427.222,171.615,29.508,155.494
C01460=1059.072,45.187,427.205,171.617,29.511,155.494
C01461=1059.078,45.436,427.189,171.618,29.513,155.495
C01462=1059.085,45.721,427.170,171.620,29.516,155.495
C01463=1059.091,46.006,427.151,171.622,29.519,155.495
C01464=1059.099,46.291,427.132,171.624,29.523,155.496
C01465=1059.106,46.576,427.113,171.625,29.525,155.496
C01466=1059.112,46.826,427.096,171.626,29.528,155.497
C01467=1059.117,47.075,427.080,171.628,29.530,155.497
C01468=1059.123,47.325,427.063,171.629,29.533,155.497
C01469=1059.130,47.574,427.046,171.631,29.536,155.498
C01470=1059.135,47.824,427.029,171.632,29.538,155.498
C01471=1059.141,48.073,427.013,171.633,29.540,155.499
C01472=1059.147,48.322,426.996,171.635,29.543,155.499
C01473=1059.153,48.571,426.980,171.637,29.546,155.499
C01474=1059.159,48.821,426.962,171.638,29.548,155.500
C01475=1059.165,49.070,426.945,171.639,29.550,155.500
C01476=1059.171,49.320,426.929,171.641,29.553,155.500
C01477=1059.177,49.569,426.912,171.643,29.555,155.501
C01478=1059.182,49.818,426.895,171.643,29.558,155.501
C01479=1059.189,50.067,426.878,171.645,29.561,155.502
C01480=1059.195,50.317,426.862,171.647,29.563,155.502
C01481=1059.201,50.566,426.845,171.649,29.566,155.502
C01482=1059.207,50.815,426.828,171.650,29.568,155.503
C01483=1059.213,51.065,426.811,171.651,29.570,155.503
C01484=1059.219,51.314,426.794,171.653,29.573,155.503
C01485=1059.225,51.564,426.777,171.654,29.576,155.504
C01486=1059.232,51.813,426.760,171.656,29.579,155.504
C01487=1059.237,52.063,426.743,171.657,29.581,155.504
C01488=1059.243,52.311,426.726,171.659,29.583,155.505
C01489=1059.249,52.561,426.710,171.660,29.586,155.505
C01490=1059.255,52.811,426.693,171.662,29.588,155.506
C01491=1059.261,53.060,426.676,171.663,29.591,155.506
C01492=1059.267,53.309,426.660,171.664,29.594,155.506
C01493=1059.273,53.559,426.642,171.666,29.596,155.507
C01494=1059.279,53.808,426.625,171.668,29.598,155.507
C01495=1059.285,54.057,426.608,171.669,29.601,155.507
C01496=1059.292,54.307,426.591,171.670,29.603,155.508
C01497=1059.297,54.556,426.574,171.672,29.606,155.508
C01498=1059.304,54.805,426.557,171.674,29.609,155.509
C01499=1059.310,55.055,426.540,171.676,29.611,155.509
C01500=1059.316,55.304,426.523,171.676,29.613,155.509
C01501=1059.322,55.553,426.507,171.678,29.616,155.510
C01502=1059.328,55.803,426.489,171.680,29.618,155.510
C01503=1059.334,56.052,426.472,171.681,29.621,155.510
C01504=1059.339,56.301,426.455,171.682,29.624,155.511
C01505=1059.346,56.551,426.438,171.684,29.626,155.511
C01506=1059.352,56.800,426.422,171.686,29.629,155.511
C01507=1059.358,57.049,426.404,171.687,29.631,155.512
C01508=1059.365,57.299,426.387,171.688,29.633,155.512
C01509=1059.370,57.548,426.370,171.690,29.636,155.513
C01510=1059.377,57.798,426.352,171.691,29.639,155.513
C01511=1059.383,58.046,426.335,171.693,29.641,155.513
C01512=1059.389,58.296,426.319,171.695,29.644,155.514
C01513=1059.395,58.545,426.301,171.696,29.646,155.514
C01514=1059.401,58.794,426.284,171.697,29.648,155.514
C01515=1059.407,59.045,426.267,171.699,29.651,155.515
C01516=1059.413,59.293,426.250,171.701,29.653,155.515
C01517=1059.420,59.542,426.233,171.702,29.656,155.515
C01518=1059.425,59.792,426.216,171.703,29.659,155.516
C01519=1059.432,60.041,426.199,171.705,29.661,155.516
C01520=1059.438,60.291,426.181,171.707,29.663,155.517
C01521=1059.444,60.540,426.164,171.707,29.666,155.517
C01522=1059.451,60.790,426.147,171.709,29.668,155.517
C01523=1059.456,61.039,426.130,171.711,29.671,155.518
C01524=1059.463,61.288,426.112,171.713,29.674,155.518
C01525=1059.468,61.538,426.096,171.714,29.676,155.518
C01526=1059.476,61.822,426.076,171.716,29.679,155.519
C01527=1059.483,62.106,426.056,171.718,29.681,155.519
C01528=1059.489,62.392,426.037,171.719,29.685,155.520
C01529=1059.497,62.676,426.017,171.721,29.687,155.520
C01530=1059.503,62.926,425.999,171.722,29.689,155.520
C01531=1059.509,63.174,425.982,171.724,29.692,155.521
C01532=1059.516,63.424,425.965,171.725,29.695,155.521
C01533=1059.521,63.673,425.948,171.727,29.697,155.521
C01534=1059.528,63.923,425.931,171.729,29.700,155.522
C01535=1059.534,64.172,425.913,171.729,29.702,155.522
C01536=1059.540,64.421,425.896,171.731,29.704,155.523
C01537=1059.546,64.670,425.878,171.733,29.707,155.523
C01538=1059.552,64.920,425.860,171.735,29.710,155.523
C01539=1059.558,65.169,425.844,171.735,29.712,155.524
C01540=1059.564,65.419,425.826,171.737,29.715,155.524
C01541=1059.570,65.668,425.808,171.739,29.717,155.524
C01542=1059.576,65.918,425.791,171.740,29.720,155.525
C01543=1059.582,66.167,425.773,171.741,29.722,155.525
C01544=1059.588,66.415,425.756,171.743,29.725,155.526
C01545=1059.594,66.665,425.739,171.745,29.727,155.526
C01546=1059.600,66.914,425.721,171.746,29.730,155.526
C01547=1059.607,67.164,425.704,171.747,29.732,155.527
C01548=1059.612,67.413,425.686,171.749,29.735,155.527
C01549=1059.618,67.662,425.668,171.751,29.738,155.527
C01550=1059.624,67.911,425.651,171.752,29.740,155.528
C01551=1059.631,68.161,425.633,171.754,29.743,155.528
C01552=1059.636,68.410,425.616,171.755,29.745,155.529
C01553=1059.642,68.660,425.598,171.756,29.748,155.529
C01554=1059.649,68.908,425.581,171.758,29.750,155.529
C01555=1059.655,69.158,425.563,171.760,29.753,155.530
C01556=1059.661,69.408,425.545,171.761,29.755,155.530
C01557=1059.666,69.657,425.527,171.762,29.758,155.530
C01558=1059.673,69.906,425.510,171.764,29.760,155.531
C01559=1059.679,70.155,425.492,171.766,29.763,155.531
C01560=1059.685,70.405,425.474,171.767,29.765,155.532
C01561=1059.690,70.654,425.457,171.768,29.768,155.532
C01562=1059.697,70.904,425.439,171.770,29.771,155.532
C01563=1059.702,71.153,425.421,171.772,29.773,155.533
C01564=1059.709,71.402,425.404,171.773,29.776,155.533
C01565=1059.715,71.651,425.386,171.774,29.778,155.534
C01566=1059.721,71.901,425.368,171.776,29.781,155.534
C01567=1059.726,72.150,425.350,171.778,29.784,155.534
C01568=1059.733,72.399,425.332,171.779,29.786,155.535
C01569=1059.738,72.648,425.315,171.780,29.788,155.535
C01570=1059.744,72.898,425.297,171.782,29.791,155.535
C01571=1059.751,73.148,425.280,171.784,29.794,155.536
C01572=1059.757,73.396,425.261,171.785,29.797,155.536
C01573=1059.763,73.646,425.243,171.786,29.799,155.537
C01574=1059.768,73.895,425.226,171.788,29.801,155.537
C01575=1059.775,74.144,425.208,171.789,29.804,155.537
C01576=1059.780,74.393,425.190,171.791,29.807,155.538
C01577=1059.786,74.643,425.172,171.793,29.809,155.538
C01578=1059.793,74.892,425.154,171.794,29.812,155.538
C01579=1059.798,75.141,425.136,171.795,29.814,155.539
C01580=1059.805,75.391,425.119,171.797,29.817,155.539
C01581=1059.811,75.640,425.101,171.799,29.820,155.540
C01582=1059.817,75.889,425.083,171.800,29.822,155.540
C01583=1059.823,76.139,425.065,171.801,29.824,155.540
C01584=1059.829,76.388,425.047,171.803,29.827,155.541
C01585=1059.835,76.638,425.029,171.805,29.830,155.541
C01586=1059.841,76.886,425.011,171.806,29.832,155.541
C01587=1059.847,77.136,424.993,171.807,29.835,155.542
C01588=1059.853,77.385,424.975,171.809,29.837,155.542
C01589=1059.859,77.634,424.957,171.811,29.840,155.543
C01590=1059.866,77.919,424.936,171.812,29.843,155.543
C01591=1059.873,78.204,424.916,171.814,29.845,155.543
C01592=1059.879,78.488,424.895,171.816,29.849,155.544
C01593=1059.886,78.772,424.874,171.817,29.852,155.544
C01594=1059.892,79.022,424.856,171.819,29.854,155.545
C01595=1059.898,79.271,424.839,171.820,29.857,155.545
C01596=1059.904,79.520,424.820,171.822,29.860,155.546
C01597=1059.910,79.770,424.802,171.823,29.862,155.546
C01598=1059.916,80.018,424.784,171.825,29.864,155.546
C01599=1059.922,80.268,424.766,171.827,29.867,155.547
C01600=1059.927,80.517,424.748,171.828,29.870,155.547
C01601=1059.934,80.767,424.729,171.829,29.872,155.548
C01602=1059.940,81.016,424.711,171.831,29.875,155.548
C01603=1059.946,81.265,424.693,171.833,29.878,155.548
C01604=1059.952,81.514,424.675,171.833,29.880,155.549
C01605=1059.958,81.764,424.656,171.835,29.883,155.549
C01606=1059.963,82.013,424.638,171.837,29.885,155.549
C01607=1059.969,82.262,424.620,171.839,29.888,155.550
C01608=1059.975,82.512,424.602,171.839,29.891,155.550
C01609=1059.981,82.760,424.583,171.841,29.893,155.551
C01610=1059.987,83.010,424.566,171.843,29.896,155.551
C01611=1059.994,83.259,424.547,171.845,29.899,155.552
C01612=1059.999,83.508,424.529,171.846,29.901,155.552
C01613=1060.005,83.758,424.510,171.847,29.903,155.552
C01614=1060.011,84.007,424.492,171.849,29.906,155.553
C01615=1060.017,84.256,424.474,171.851,29.909,155.553
C01616=1060.023,84.505,424.456,171.852,29.912,155.553
C01617=1060.029,84.755,424.437,171.853,29.914,155.554
C01618=1060.035,85.005,424.419,171.855,29.916,155.554
C01619=1060.041,85.253,424.400,171.856,29.919,155.555
C01620=1060.047,85.503,424.383,171.858,29.922,155.555
C01621=1060.053,85.752,424.364,171.860,29.924,155.555
C01622=1060.059,86.000,424.346,171.861,29.927,155.556
C01623=1060.064,86.250,424.327,171.862,29.929,155.556
C01624=1060.071,86.500,424.308,171.864,29.932,155.557
C01625=1060.077,86.749,424.290,171.866,29.934,155.557
C01626=1060.083,86.998,424.272,171.868,29.937,155.557
C01627=1060.089,87.247,424.254,171.868,29.940,155.558
C01628=1060.095,87.497,424.235,171.870,29.942,155.558
C01629=1060.101,87.746,424.216,171.872,29.945,155.558
C01630=1060.107,87.995,424.198,171.874,29.947,155.559
C01631=1060.113,88.244,424.180,171.875,29.950,155.559
C01632=1060.119,88.493,424.162,171.876,29.953,155.560
C01633=1060.125,88.743,424.142,171.878,29.955,155.560
C01634=1060.131,88.992,424.124,171.880,29.957,155.560
C01635=1060.137,89.241,424.106,171.881,29.960,155.561
C01636=1060.143,89.490,424.087,171.882,29.963,155.561
C01637=1060.150,89.740,424.069,171.884,29.965,155.562
C01638=1060.155,89.989,424.050,171.886,29.968,155.562
C01639=1060.162,90.238,424.032,171.887,29.970,155.562
C01640=1060.168,90.488,424.014,171.889,29.973,155.563
C01641=1060.174,90.736,423.995,171.890,29.976,155.563
C01642=1060.179,90.986,423.976,171.891,29.978,155.564
C01643=1060.186,91.235,423.957,171.893,29.981,155.564
C01644=1060.191,91.484,423.938,171.895,29.984,155.564
C01645=1060.197,91.733,423.921,171.897,29.986,155.565
C01646=1060.203,91.983,423.901,171.897,29.988,155.565
C01647=1060.209,92.232,423.883,171.899,29.991,155.565
C01648=1060.215,92.481,423.864,171.901,29.994,155.566
C01649=1060.221,92.731,423.845,171.903,29.996,155.566
C01650=1060.226,92.980,423.827,171.904,29.999,155.567
C01651=1060.232,93.229,423.808,171.905,30.002,155.567
C01652=1060.239,93.478,423.789,171.907,30.004,155.568
C01653=1060.245,93.728,423.770,171.909,30.007,155.568
C01654=1060.251,94.012,423.749,171.910,30.010,155.568
C01655=1060.258,94.297,423.727,171.912,30.013,155.569
C01656=1060.265,94.581,423.706,171.914,30.016,155.569
C01657=1060.272,94.865,423.685,171.915,30.019,155.570
C01658=1060.277,95.115,423.666,171.917,30.021,155.570
C01659=1060.283,95.364,423.647,171.919,30.024,155.570
C01660=1060.289,95.613,423.628,171.921,30.027,155.571
C01661=1060.295,95.863,423.609,171.921,30.029,155.571
C01662=1060.301,96.112,423.590,171.923,30.032,155.572
C01663=1060.308,96.361,423.572,171.925,30.035,155.572
C01664=1060.313,96.610,423.553,171.927,30.037,155.572
C01665=1060.319,96.859,423.534,171.928,30.040,155.573
C01666=1060.325,97.108,423.515,171.929,30.042,155.573
C01667=1060.331,97.357,423.496,171.931,30.045,155.574
C01668=1060.337,97.607,423.477,171.933,30.048,155.574
C01669=1060.343,97.856,423.458,171.934,30.050,155.574
C01670=1060.349,98.105,423.439,171.936,30.053,155.575
C01671=1060.355,98.355,423.420,171.937,30.055,155.575
C01672=1060.361,98.604,423.401,171.939,30.058,155.576
C01673=1060.368,98.853,423.383,171.940,30.060,155.576
C01674=1060.373,99.102,423.364,171.942,30.063,155.576
C01675=1060.379,99.351,423.345,171.944,30.066,155.577
C01676=1060.385,99.600,423.326,171.945,30.068,155.577
C01677=1060.391,99.850,423.307,171.946,30.071,155.578
C01678=1060.397,100.099,423.288,171.948,30.074,155.578
C01679=1060.403,100.348,423.269,171.950,30.076,155.578
C01680=1060.409,100.598,423.250,171.952,30.079,155.579
C01681=1060.415,100.847,423.231,171.953,30.081,155.579
C01682=1060.421,101.095,423.211,171.954,30.084,155.580
C01683=1060.427,101.345,423.192,171.956,30.086,155.580
C01684=1060.433,101.594,423.173,171.957,30.089,155.580
C01685=1060.439,101.843,423.154,171.959,30.092,155.581
C01686=1060.445,102.093,423.135,171.961,30.095,155.581
C01687=1060.451,102.342,423.116,171.962,30.097,155.582
C01688=1060.456,102.591,423.097,171.963,30.100,155.582
C01689=1060.462,102.840,423.077,171.965,30.103,155.582
C01690=1060.468,103.089,423.058,171.967,30.105,155.583
C01691=1060.474,103.338,423.039,171.969,30.107,155.583
C01692=1060.479,103.588,423.020,171.970,30.110,155.584
C01693=1060.486,103.837,423.001,171.971,30.113,155.584
C01694=1060.492,104.086,422.981,171.973,30.115,155.584
C01695=1060.498,104.335,422.962,171.975,30.118,155.585
C01696=1060.503,104.585,422.943,171.976,30.121,155.585
C01697=1060.509,104.834,422.923,171.978,30.123,155.586
C01698=1060.515,105.083,422.905,171.979,30.126,155.586
C01699=1060.521,105.332,422.885,171.981,30.129,155.586
C01700=1060.527,105.581,422.866,171.982,30.131,155.587
C01701=1060.533,105.831,422.846,171.984,30.134,155.587
C01702=1060.539,106.079,422.827,171.986,30.137,155.588
C01703=1060.545,106.329,422.808,171.988,30.139,155.588
C01704=1060.551,106.578,422.788,171.988,30.142,155.588
C01705=1060.557,106.828,422.769,171.990,30.144,155.589
C01706=1060.563,107.077,422.749,171.992,30.147,155.589
C01707=1060.569,107.326,422.731,171.994,30.149,155.590
C01708=1060.575,107.575,422.711,171.995,30.152,155.590
C01709=1060.581,107.824,422.691,171.997,30.155,155.590
C01710=1060.586,108.073,422.672,171.998,30.157,155.591
C01711=1060.592,108.323,422.653,172.000,30.160,155.591
C01712=1060.599,108.571,422.634,172.001,30.163,155.592
C01713=1060.604,108.821,422.614,172.003,30.166,155.592
C01714=1060.610,109.069,422.594,172.005,30.168,155.592
C01715=1060.616,109.319,422.575,172.007,30.170,155.593
C01716=1060.622,109.568,422.556,172.007,30.173,155.593
C01717=1060.629,109.817,422.537,172.009,30.176,155.594
C01718=1060.635,110.102,422.515,172.011,30.179,155.594
C01719=1060.643,110.386,422.492,172.014,30.182,155.594
C01720=1060.648,110.671,422.470,172.015,30.184,155.595
C01721=1060.655,110.955,422.447,172.017,30.188,155.595
C01722=1060.662,111.204,422.428,172.019,30.190,155.596
C01723=1060.668,111.453,422.408,172.020,30.193,155.596
C01724=1060.673,111.703,422.389,172.021,30.196,155.597
C01725=1060.680,111.952,422.369,172.023,30.198,155.597
C01726=1060.686,112.201,422.350,172.025,30.201,155.597
C01727=1060.692,112.450,422.330,172.027,30.203,155.598
C01728=1060.697,112.700,422.310,172.028,30.206,155.598
C01729=1060.703,112.949,422.290,172.030,30.209,155.599
C01730=1060.709,113.198,422.271,172.031,30.211,155.599
C01731=1060.715,113.447,422.251,172.033,30.214,155.599
C01732=1060.721,113.696,422.232,172.034,30.216,155.600
C01733=1060.727,113.945,422.212,172.036,30.219,155.600
C01734=1060.732,114.194,422.193,172.038,30.222,155.601
C01735=1060.738,114.443,422.173,172.040,30.225,155.601
C01736=1060.744,114.693,422.154,172.041,30.227,155.601
C01737=1060.749,114.942,422.133,172.042,30.230,155.602
C01738=1060.756,115.191,422.113,172.044,30.232,155.602
C01739=1060.762,115.441,422.093,172.046,30.235,155.603
C01740=1060.767,115.690,422.073,172.047,30.238,155.603
C01741=1060.773,115.938,422.053,172.049,30.241,155.604
C01742=1060.778,116.188,422.034,172.051,30.243,155.604
C01743=1060.784,116.437,422.014,172.052,30.246,155.604
C01744=1060.790,116.686,421.994,172.053,30.248,155.605
C01745=1060.796,116.935,421.974,172.055,30.251,155.605
C01746=1060.802,117.184,421.955,172.057,30.254,155.606
C01747=1060.807,117.433,421.934,172.059,30.257,155.606
C01748=1060.813,117.683,421.915,172.060,30.260,155.607
C01749=1060.819,117.931,421.895,172.062,30.263,155.607
C01750=1060.826,118.181,421.874,172.063,30.265,155.607
C01751=1060.831,118.430,421.855,172.065,30.268,155.608
C01752=1060.837,118.679,421.835,172.066,30.270,155.608
C01753=1060.843,118.928,421.815,172.068,30.273,155.609
C01754=1060.849,119.177,421.795,172.070,30.276,155.609
C01755=1060.854,119.427,421.775,172.072,30.279,155.609
C01756=1060.860,119.676,421.755,172.073,30.281,155.610
C01757=1060.866,119.925,421.735,172.075,30.284,155.610
C01758=1060.872,120.174,421.715,172.076,30.286,155.611
C01759=1060.878,120.423,421.695,172.078,30.289,155.611
C01760=1060.883,120.673,421.675,172.079,30.292,155.611
C01761=1060.889,120.921,421.655,172.081,30.294,155.612
C01762=1060.895,121.170,421.635,172.083,30.297,155.612
C01763=1060.902,121.420,421.615,172.085,30.300,155.613
C01764=1060.907,121.669,421.594,172.086,30.303,155.613
C01765=1060.913,121.918,421.574,172.088,30.305,155.614
C01766=1060.919,122.167,421.555,172.089,30.308,155.614
C01767=1060.925,122.416,421.535,172.091,30.310,155.614
C01768=1060.930,122.666,421.514,172.092,30.313,155.615
C01769=1060.936,122.914,421.494,172.094,30.316,155.615
C01770=1060.942,123.163,421.474,172.096,30.319,155.616
C01771=1060.948,123.412,421.454,172.098,30.321,155.616
C01772=1060.954,123.661,421.434,172.099,30.324,155.616
C01773=1060.960,123.911,421.413,172.101,30.326,155.617
C01774=1060.966,124.160,421.393,172.103,30.329,155.617
C01775=1060.972,124.409,421.374,172.104,30.331,155.618
C01776=1060.977,124.658,421.353,172.106,30.334,155.618
C01777=1060.984,124.908,421.333,172.107,30.337,155.618
C01778=1060.990,125.156,421.313,172.109,30.339,155.619
C01779=1060.995,125.406,421.293,172.111,30.342,155.619
C01780=1061.001,125.654,421.273,172.113,30.345,155.620
C01781=1061.008,125.904,421.252,172.114,30.347,155.620
C01782=1061.014,126.189,421.229,172.116,30.351,155.621
C01783=1061.021,126.472,421.206,172.118,30.353,155.621
C01784=1061.028,126.757,421.182,172.120,30.357,155.621
C01785=1061.035,127.041,421.160,172.122,30.359,155.622
C01786=1061.040,127.290,421.139,172.123,30.362,155.622
C01787=1061.046,127.539,421.119,172.125,30.365,155.623
C01788=1061.053,127.789,421.099,172.127,30.367,155.623
C01789=1061.058,128.038,421.078,172.128,30.370,155.624
C01790=1061.064,128.287,421.058,172.130,30.373,155.624
C01791=1061.071,128.536,421.038,172.132,30.375,155.624
C01792=1061.076,128.785,421.017,172.134,30.378,155.625
C01793=1061.082,129.034,420.997,172.135,30.381,155.625
C01794=1061.089,129.284,420.977,172.137,30.383,155.626
C01795=1061.094,129.532,420.956,172.139,30.386,155.626
C01796=1061.100,129.781,420.936,172.141,30.389,155.626
C01797=1061.107,130.031,420.916,172.142,30.391,155.627
C01798=1061.112,130.280,420.895,172.144,30.394,155.627
C01799=1061.118,130.528,420.875,172.145,30.396,155.628
C01800=1061.125,130.778,420.855,172.147,30.399,155.628
C01801=1061.130,131.027,420.834,172.149,30.401,155.628
C01802=1061.136,131.277,420.814,172.150,30.404,155.629
C01803=1061.143,131.525,420.793,172.152,30.407,155.629
C01804=1061.148,131.774,420.773,172.154,30.409,155.630
C01805=1061.155,132.023,420.752,172.156,30.412,155.630
C01806=1061.160,132.273,420.732,172.157,30.415,155.630
C01807=1061.166,132.521,420.711,172.159,30.418,155.631
C01808=1061.172,132.771,420.690,172.161,30.420,155.631
C01809=1061.177,133.020,420.670,172.163,30.423,155.632
C01810=1061.183,133.269,420.650,172.164,30.426,155.632
C01811=1061.189,133.518,420.628,172.166,30.428,155.632
C01812=1061.195,133.767,420.608,172.168,30.431,155.633
C01813=1061.201,134.016,420.588,172.170,30.434,155.633
C01814=1061.207,134.266,420.567,172.171,30.436,155.634
C01815=1061.213,134.514,420.546,172.172,30.439,155.634
C01816=1061.219,134.764,420.525,172.174,30.441,155.635
C01817=1061.225,135.012,420.505,172.176,30.444,155.635
C01818=1061.230,135.261,420.484,172.178,30.447,155.635
C01819=1061.236,135.511,420.463,172.179,30.450,155.636
